LIN {X 0,Y 320.102,Z 625.92,A -85,B 0,C 180,E1 2193.671,E2 2193.671} C_VEL
LIN {X 0,Y 317.839,Z 623.977,A -85,B 0,C 180,E1 2191.692,E2 2191.692} C_VEL
LIN {X 0,Y 312.964,Z 620.611,A -85,B 0,C 180,E1 2187.803,E2 2187.803} C_VEL
LIN {X 0,Y 308.078,Z 616.466,A -85,B 0,C 180,E1 2184.137,E2 2184.137} C_VEL
LIN {X 0,Y 302.744,Z 613.332,A -85,B 0,C 180,E1 2180.694,E2 2180.694} C_VEL
LIN {X 0,Y 290.783,Z 600.623,A -85,B 0,C 180,E1 2170,E2 2170} C_VEL
LIN {X 0,Y 289.922,Z 598.567,A -85,B 0,C 180,E1 2168.424,E2 2168.424} C_VEL
LIN {X 0,Y 284.718,Z 621.095,A -85,B 0,C 180,E1 2168.26,E2 2168.26} C_VEL
LIN {X 0,Y 277.743,Z 643.252,A -85,B 0,C 180,E1 2168.127,E2 2168.127} C_VEL
LIN {X 0,Y 269.048,Z 664.747,A -85,B 0,C 180,E1 2167.961,E2 2167.961} C_VEL
LIN {X 0,Y 258.806,Z 685.28,A -85,B 0,C 180,E1 2167.727,E2 2167.727} C_VEL
LIN {X 0,Y 246.51,Z 705.546,A -85,B 0,C 180,E1 2167.398,E2 2167.398} C_VEL
LIN {X 0,Y 233.192,Z 724.08,A -85,B 0,C 180,E1 2166.987,E2 2166.987} C_VEL
LIN {X 0,Y 217.831,Z 742.232,A -85,B 0,C 180,E1 2166.425,E2 2166.425} C_VEL
LIN {X 0,Y 201.977,Z 758.277,A -85,B 0,C 180,E1 2165.734,E2 2165.734} C_VEL
LIN {X 0,Y 183.6,Z 774.186,A -85,B 0,C 180,E1 2164.75,E2 2164.75} C_VEL
LIN {X 0,Y 165.285,Z 787.803,A -85,B 0,C 180,E1 2163.525,E2 2163.525} C_VEL
LIN {X 0,Y 145.045,Z 800.516,A -85,B 0,C 180,E1 2161.78,E2 2161.78} C_VEL
LIN {X 0,Y 125.982,Z 810.635,A -85,B 0,C 180,E1 2159.595,E2 2159.595} C_VEL
LIN {X 0,Y 104.228,Z 820.309,A -85,B 0,C 180,E1 2156.063,E2 2156.063} C_VEL
LIN {X 0,Y 84.008,Z 827.603,A -85,B 0,C 180,E1 2151.055,E2 2151.055} C_VEL
LIN {X 0,Y 63.033,Z 833.661,A -85,B 0,C 180,E1 2142.124,E2 2142.124} C_VEL
LIN {X 0,Y 45.429,Z 837.544,A -85,B 0,C 180,E1 2126.617,E2 2126.617} C_VEL
LIN {X 0,Y 34.523,Z 839.63,A -85,B 0,C 180,E1 2101.419,E2 2101.419} C_VEL
LIN {X 0,Y 32.041,Z 840.272,A -85,B 0,C 180,E1 2073.061,E2 2073.061} C_VEL
LIN {X 0,Y 32.169,Z 840.12,A -85,B 0,C 180,E1 2057.434,E2 2057.434} C_VEL
LIN {X 0,Y 37.039,Z 839.124,A -85,B 0,C 180,E1 2029.62,E2 2029.62} C_VEL
LIN {X 0,Y 51.419,Z 836.361,A -85,B 0,C 180,E1 2006.561,E2 2006.561} C_VEL
LIN {X 0,Y 70.128,Z 831.753,A -85,B 0,C 180,E1 1994.188,E2 1994.188} C_VEL
LIN {X 0,Y 89.711,Z 825.717,A -85,B 0,C 180,E1 1987.293,E2 1987.293} C_VEL
LIN {X 0,Y 111.668,Z 817.214,A -85,B 0,C 180,E1 1982.566,E2 1982.566} C_VEL
LIN {X 0,Y 129.978,Z 808.641,A -85,B 0,C 180,E1 1979.893,E2 1979.893} C_VEL
LIN {X 0,Y 150.342,Z 797.394,A -85,B 0,C 180,E1 1977.713,E2 1977.713} C_VEL
LIN {X 0,Y 169.348,Z 784.933,A -85,B 0,C 180,E1 1976.176,E2 1976.176} C_VEL
LIN {X 0,Y 187.678,Z 770.939,A -85,B 0,C 180,E1 1975.014,E2 1975.014} C_VEL
LIN {X 0,Y 205.046,Z 755.352,A -85,B 0,C 180,E1 1974.123,E2 1974.123} C_VEL
LIN {X 0,Y 220.902,Z 738.824,A -85,B 0,C 180,E1 1973.455,E2 1973.455} C_VEL
LIN {X 0,Y 235.753,Z 720.694,A -85,B 0,C 180,E1 1972.929,E2 1972.929} C_VEL
LIN {X 0,Y 249.072,Z 701.604,A -85,B 0,C 180,E1 1972.53,E2 1972.53} C_VEL
LIN {X 0,Y 251.814,Z 697.259,A -85,B 0,C 180,E1 1972.457,E2 1972.457} C_VEL
LIN {X 0,Y 255.871,Z 690.789,A -85,B 0,C 180,E1 1972.136,E2 1972.136} C_VEL
LIN {X 0,Y 265.428,Z 674.452,A -85,B 0,C 180,E1 1970.638,E2 1970.638} C_VEL
LIN {X 0,Y 268.838,Z 667.606,A -85,B 0,C 180,E1 1970.369,E2 1970.369} C_VEL
LIN {X 0,Y 277.455,Z 647.28,A -85,B 0,C 180,E1 1970.258,E2 1970.258} C_VEL
LIN {X 0,Y 285.113,Z 624.081,A -85,B 0,C 180,E1 1970.163,E2 1970.163} C_VEL
LIN {X 0,Y 289.087,Z 608.609,A -85,B 0,C 180,E1 1970.042,E2 1970.042} C_VEL
LIN {X 0,Y 301.141,Z 621.43,A -85,B 0,C 180,E1 1958.987,E2 1958.987} C_VEL
LIN {X 0,Y 306.567,Z 624.761,A -85,B 0,C 180,E1 1955.428,E2 1955.428} C_VEL
LIN {X 0,Y 311.119,Z 628.561,A -85,B 0,C 180,E1 1952.017,E2 1952.017} C_VEL
LIN {X 0,Y 315.891,Z 631.757,A -85,B 0,C 180,E1 1948.303,E2 1948.303} C_VEL
LIN {X 0,Y 318.81,Z 634.401,A -85,B 0,C 180,E1 1945.74,E2 1945.74} C_VEL
LIN {X 0,Y 322.94,Z 637.822,A -85,B 0,C 180,E1 1941.966,E2 1941.966} C_VEL
LIN {X 0,Y 327.018,Z 640.577,A -85,B 0,C 180,E1 1938.082,E2 1938.082} C_VEL
LIN {X 0,Y 330.44,Z 644.079,A -85,B 0,C 180,E1 1934.343,E2 1934.343} C_VEL
LIN {X 0,Y 333.893,Z 646.67,A -85,B 0,C 180,E1 1930.482,E2 1930.482} C_VEL
LIN {X 0,Y 336.83,Z 648.45,A -85,B 0,C 180,E1 1927.012,E2 1927.012} C_VEL
LIN {X 0,Y 339.519,Z 651.579,A -85,B 0,C 180,E1 1923.212,E2 1923.212} C_VEL
LIN {X 0,Y 342.103,Z 653.743,A -85,B 0,C 180,E1 1919.406,E2 1919.406} C_VEL
LIN {X 0,Y 344.514,Z 655.168,A -85,B 0,C 180,E1 1915.499,E2 1915.499} C_VEL
LIN {X 0,Y 346.58,Z 656.053,A -85,B 0,C 180,E1 1911.729,E2 1911.729} C_VEL
LIN {X 0,Y 348.102,Z 658.201,A -85,B 0,C 180,E1 1907.898,E2 1907.898} C_VEL
LIN {X 0,Y 349.354,Z 659.732,A -85,B 0,C 180,E1 1904.248,E2 1904.248} C_VEL
LIN {X 0,Y 350.337,Z 660.737,A -85,B 0,C 180,E1 1900.524,E2 1900.524} C_VEL
LIN {X 0,Y 351.081,Z 661.354,A -85,B 0,C 180,E1 1896.705,E2 1896.705} C_VEL
LIN {X 0,Y 351.475,Z 661.618,A -85,B 0,C 180,E1 1893.135,E2 1893.135} C_VEL
LIN {X 0,Y 351.583,Z 661.704,A -85,B 0,C 180,E1 1889.348,E2 1889.348} C_VEL
LIN {X 0,Y 351.381,Z 661.597,A -85,B 0,C 180,E1 1885.921,E2 1885.921} C_VEL
LIN {X 0,Y 350.894,Z 661.181,A -85,B 0,C 180,E1 1882.139,E2 1882.139} C_VEL
LIN {X 0,Y 350.09,Z 660.488,A -85,B 0,C 180,E1 1878.409,E2 1878.409} C_VEL
LIN {X 0,Y 349.022,Z 659.363,A -85,B 0,C 180,E1 1874.719,E2 1874.719} C_VEL
LIN {X 0,Y 347.649,Z 657.577,A -85,B 0,C 180,E1 1870.861,E2 1870.861} C_VEL
LIN {X 0,Y 346.392,Z 655.984,A -85,B 0,C 180,E1 1867.905,E2 1867.905} C_VEL
LIN {X 0,Y 344.411,Z 655.129,A -85,B 0,C 180,E1 1864.371,E2 1864.371} C_VEL
LIN {X 0,Y 341.976,Z 653.652,A -85,B 0,C 180,E1 1860.389,E2 1860.389} C_VEL
LIN {X 0,Y 339.315,Z 651.382,A -85,B 0,C 180,E1 1856.503,E2 1856.503} C_VEL
LIN {X 0,Y 336.812,Z 648.412,A -85,B 0,C 180,E1 1852.943,E2 1852.943} C_VEL
LIN {X 0,Y 333.403,Z 646.352,A -85,B 0,C 180,E1 1848.947,E2 1848.947} C_VEL
LIN {X 0,Y 330.101,Z 643.814,A -85,B 0,C 180,E1 1845.356,E2 1845.356} C_VEL
LIN {X 0,Y 327.244,Z 640.903,A -85,B 0,C 180,E1 1842.236,E2 1842.236} C_VEL
LIN {X 0,Y 325.416,Z 639.465,A -85,B 0,C 180,E1 1840.362,E2 1840.362} C_VEL
LIN {X 0,Y 321.239,Z 636.539,A -85,B 0,C 180,E1 1836.476,E2 1836.476} C_VEL
LIN {X 0,Y 317.034,Z 632.556,A -85,B 0,C 180,E1 1832.636,E2 1832.636} C_VEL
LIN {X 0,Y 312.081,Z 629.265,A -85,B 0,C 180,E1 1828.723,E2 1828.723} C_VEL
LIN {X 0,Y 307.338,Z 625.454,A -85,B 0,C 180,E1 1825.122,E2 1825.122} C_VEL
LIN {X 0,Y 304.559,Z 623.461,A -85,B 0,C 180,E1 1823.201,E2 1823.201} C_VEL
LIN {X 0,Y 298.441,Z 619.537,A -85,B 0,C 180,E1 1819.269,E2 1819.269} C_VEL
LIN {X 0,Y 291.516,Z 612.567,A -85,B 0,C 180,E1 1813.285,E2 1813.285} C_VEL
LIN {X 0,Y 289.022,Z 608.749,A -85,B 0,C 180,E1 1809.919,E2 1809.919} C_VEL
LIN {X 0,Y 282.774,Z 631.763,A -85,B 0,C 180,E1 1809.809,E2 1809.809} C_VEL
LIN {X 0,Y 274.898,Z 653.734,A -85,B 0,C 180,E1 1809.717,E2 1809.717} C_VEL
LIN {X 0,Y 265.662,Z 674.23,A -85,B 0,C 180,E1 1809.583,E2 1809.583} C_VEL
LIN {X 0,Y 255.391,Z 693.035,A -85,B 0,C 180,E1 1809.406,E2 1809.406} C_VEL
LIN {X 0,Y 242.675,Z 712.598,A -85,B 0,C 180,E1 1809.148,E2 1809.148} C_VEL
LIN {X 0,Y 228.664,Z 730.782,A -85,B 0,C 180,E1 1808.817,E2 1808.817} C_VEL
LIN {X 0,Y 213.039,Z 748.159,A -85,B 0,C 180,E1 1808.366,E2 1808.366} C_VEL
LIN {X 0,Y 196.79,Z 763.614,A -85,B 0,C 180,E1 1807.806,E2 1807.806} C_VEL
LIN {X 0,Y 180.354,Z 777.15,A -85,B 0,C 180,E1 1807.104,E2 1807.104} C_VEL
LIN {X 0,Y 160.873,Z 790.935,A -85,B 0,C 180,E1 1806.065,E2 1806.065} C_VEL
LIN {X 0,Y 140.436,Z 803.092,A -85,B 0,C 180,E1 1804.64,E2 1804.64} C_VEL
LIN {X 0,Y 119.102,Z 813.711,A -85,B 0,C 180,E1 1802.598,E2 1802.598} C_VEL
LIN {X 0,Y 98.984,Z 821.939,A -85,B 0,C 180,E1 1799.842,E2 1799.842} C_VEL
LIN {X 0,Y 77.255,Z 829.128,A -85,B 0,C 180,E1 1795.222,E2 1795.222} C_VEL
LIN {X 0,Y 56.371,Z 834.404,A -85,B 0,C 180,E1 1787.294,E2 1787.294} C_VEL
LIN {X 0,Y 38.335,Z 837.829,A -85,B 0,C 180,E1 1772.469,E2 1772.469} C_VEL
LIN {X 0,Y 25.468,Z 839.709,A -85,B 0,C 180,E1 1738.106,E2 1738.106} C_VEL
LIN {X 0,Y 24.077,Z 840.061,A -85,B 0,C 180,E1 1710,E2 1710} C_VEL
LIN {X 0,Y 26.34,Z 839.628,A -85,B 0,C 180,E1 1676.629,E2 1676.629} C_VEL
LIN {X 0,Y 39.907,Z 837.567,A -85,B 0,C 180,E1 1645.587,E2 1645.587} C_VEL
LIN {X 0,Y 58.213,Z 834.008,A -85,B 0,C 180,E1 1631.765,E2 1631.765} C_VEL
LIN {X 0,Y 80.183,Z 828.281,A -85,B 0,C 180,E1 1624.009,E2 1624.009} C_VEL
LIN {X 0,Y 101.984,Z 820.822,A -85,B 0,C 180,E1 1619.678,E2 1619.678} C_VEL
LIN {X 0,Y 124.166,Z 811.372,A -85,B 0,C 180,E1 1616.851,E2 1616.851} C_VEL
LIN {X 0,Y 143.496,Z 801.397,A -85,B 0,C 180,E1 1615.12,E2 1615.12} C_VEL
LIN {X 0,Y 162.922,Z 789.581,A -85,B 0,C 180,E1 1613.812,E2 1613.812} C_VEL
LIN {X 0,Y 182.408,Z 775.547,A -85,B 0,C 180,E1 1612.799,E2 1612.799} C_VEL
LIN {X 0,Y 200.186,Z 760.621,A -85,B 0,C 180,E1 1612.067,E2 1612.067} C_VEL
LIN {X 0,Y 217.352,Z 743.64,A -85,B 0,C 180,E1 1611.498,E2 1611.498} C_VEL
LIN {X 0,Y 232.362,Z 726.314,A -85,B 0,C 180,E1 1611.089,E2 1611.089} C_VEL
LIN {X 0,Y 246.142,Z 707.607,A -85,B 0,C 180,E1 1610.776,E2 1610.776} C_VEL
LIN {X 0,Y 257.962,Z 688.601,A -85,B 0,C 180,E1 1610.544,E2 1610.544} C_VEL
LIN {X 0,Y 268.838,Z 667.606,A -85,B 0,C 180,E1 1610.369,E2 1610.369} C_VEL
LIN {X 0,Y 272.169,Z 660.669,A -85,B 0,C 180,E1 1610.127,E2 1610.127} C_VEL
LIN {X 0,Y 280.144,Z 643.301,A -85,B 0,C 180,E1 1608.817,E2 1608.817} C_VEL
LIN {X 0,Y 282.804,Z 636.101,A -85,B 0,C 180,E1 1608.603,E2 1608.603} C_VEL
LIN {X 0,Y 288.084,Z 618.389,A -85,B 0,C 180,E1 1608.544,E2 1608.544} C_VEL
LIN {X 0,Y 292.739,Z 624.151,A -85,B 0,C 180,E1 1603.429,E2 1603.429} C_VEL
LIN {X 0,Y 301.039,Z 630.48,A -85,B 0,C 180,E1 1597.545,E2 1597.545} C_VEL
LIN {X 0,Y 304.376,Z 632.619,A -85,B 0,C 180,E1 1595.343,E2 1595.343} C_VEL
LIN {X 0,Y 309.353,Z 636.641,A -85,B 0,C 180,E1 1591.633,E2 1591.633} C_VEL
LIN {X 0,Y 314.36,Z 639.845,A -85,B 0,C 180,E1 1587.781,E2 1587.781} C_VEL
LIN {X 0,Y 318.543,Z 643.821,A -85,B 0,C 180,E1 1584.058,E2 1584.058} C_VEL
LIN {X 0,Y 322.898,Z 646.911,A -85,B 0,C 180,E1 1580.135,E2 1580.135} C_VEL
LIN {X 0,Y 325.225,Z 648.595,A -85,B 0,C 180,E1 1577.917,E2 1577.917} C_VEL
LIN {X 0,Y 328.789,Z 652.073,A -85,B 0,C 180,E1 1574.137,E2 1574.137} C_VEL
LIN {X 0,Y 332.304,Z 654.586,A -85,B 0,C 180,E1 1570.307,E2 1570.307} C_VEL
LIN {X 0,Y 335.15,Z 656.305,A -85,B 0,C 180,E1 1567.057,E2 1567.057} C_VEL
LIN {X 0,Y 337.799,Z 659.322,A -85,B 0,C 180,E1 1563.403,E2 1563.403} C_VEL
LIN {X 0,Y 340.461,Z 661.535,A -85,B 0,C 180,E1 1559.562,E2 1559.562} C_VEL
LIN {X 0,Y 342.896,Z 662.969,A -85,B 0,C 180,E1 1555.751,E2 1555.751} C_VEL
LIN {X 0,Y 345.097,Z 663.894,A -85,B 0,C 180,E1 1551.947,E2 1551.947} C_VEL
LIN {X 0,Y 346.625,Z 665.9,A -85,B 0,C 180,E1 1548.325,E2 1548.325} C_VEL
LIN {X 0,Y 347.922,Z 667.484,A -85,B 0,C 180,E1 1544.648,E2 1544.648} C_VEL
LIN {X 0,Y 348.994,Z 668.566,A -85,B 0,C 180,E1 1540.899,E2 1540.899} C_VEL
LIN {X 0,Y 349.798,Z 669.201,A -85,B 0,C 180,E1 1537.06,E2 1537.06} C_VEL
LIN {X 0,Y 350.268,Z 669.523,A -85,B 0,C 180,E1 1533.273,E2 1533.273} C_VEL
LIN {X 0,Y 350.374,Z 669.619,A -85,B 0,C 180,E1 1529.509,E2 1529.509} C_VEL
LIN {X 0,Y 350.147,Z 669.5,A -85,B 0,C 180,E1 1525.906,E2 1525.906} C_VEL
LIN {X 0,Y 349.635,Z 669.089,A -85,B 0,C 180,E1 1522.276,E2 1522.276} C_VEL
LIN {X 0,Y 348.813,Z 668.434,A -85,B 0,C 180,E1 1518.593,E2 1518.593} C_VEL
LIN {X 0,Y 347.755,Z 667.302,A -85,B 0,C 180,E1 1514.833,E2 1514.833} C_VEL
LIN {X 0,Y 346.421,Z 665.635,A -85,B 0,C 180,E1 1511.14,E2 1511.14} C_VEL
LIN {X 0,Y 345.072,Z 663.886,A -85,B 0,C 180,E1 1508.004,E2 1508.004} C_VEL
LIN {X 0,Y 342.801,Z 662.921,A -85,B 0,C 180,E1 1504.056,E2 1504.056} C_VEL
LIN {X 0,Y 340.303,Z 661.435,A -85,B 0,C 180,E1 1500.229,E2 1500.229} C_VEL
LIN {X 0,Y 337.633,Z 659.166,A -85,B 0,C 180,E1 1496.375,E2 1496.375} C_VEL
LIN {X 0,Y 334.789,Z 655.876,A -85,B 0,C 180,E1 1492.466,E2 1492.466} C_VEL
LIN {X 0,Y 331.341,Z 653.985,A -85,B 0,C 180,E1 1488.636,E2 1488.636} C_VEL
LIN {X 0,Y 327.939,Z 651.333,A -85,B 0,C 180,E1 1484.982,E2 1484.982} C_VEL
LIN {X 0,Y 324.58,Z 647.915,A -85,B 0,C 180,E1 1481.475,E2 1481.475} C_VEL
LIN {X 0,Y 320.732,Z 645.471,A -85,B 0,C 180,E1 1477.889,E2 1477.889} C_VEL
LIN {X 0,Y 316.383,Z 641.914,A -85,B 0,C 180,E1 1474.012,E2 1474.012} C_VEL
LIN {X 0,Y 313.673,Z 639.451,A -85,B 0,C 180,E1 1471.673,E2 1471.673} C_VEL
LIN {X 0,Y 308.376,Z 635.921,A -85,B 0,C 180,E1 1467.623,E2 1467.623} C_VEL
LIN {X 0,Y 303.057,Z 631.562,A -85,B 0,C 180,E1 1463.735,E2 1463.735} C_VEL
LIN {X 0,Y 297.543,Z 628.3,A -85,B 0,C 180,E1 1460.25,E2 1460.25} C_VEL
LIN {X 0,Y 288.077,Z 618.375,A -85,B 0,C 180,E1 1451.445,E2 1451.445} C_VEL
LIN {X 0,Y 280.983,Z 641.308,A -85,B 0,C 180,E1 1451.386,E2 1451.386} C_VEL
LIN {X 0,Y 272.778,Z 662,A -85,B 0,C 180,E1 1451.338,E2 1451.338} C_VEL
LIN {X 0,Y 263.015,Z 681.892,A -85,B 0,C 180,E1 1451.255,E2 1451.255} C_VEL
LIN {X 0,Y 250.661,Z 702.717,A -85,B 0,C 180,E1 1451.116,E2 1451.116} C_VEL
LIN {X 0,Y 237.784,Z 720.866,A -85,B 0,C 180,E1 1450.943,E2 1450.943} C_VEL
LIN {X 0,Y 222.317,Z 739.456,A -85,B 0,C 180,E1 1450.684,E2 1450.684} C_VEL
LIN {X 0,Y 205.993,Z 756.147,A -85,B 0,C 180,E1 1450.346,E2 1450.346} C_VEL
LIN {X 0,Y 187.747,Z 772.052,A -85,B 0,C 180,E1 1449.87,E2 1449.87} C_VEL
LIN {X 0,Y 169.173,Z 785.863,A -85,B 0,C 180,E1 1449.253,E2 1449.253} C_VEL
LIN {X 0,Y 148.553,Z 798.868,A -85,B 0,C 180,E1 1448.36,E2 1448.36} C_VEL
LIN {X 0,Y 128.146,Z 809.543,A -85,B 0,C 180,E1 1447.171,E2 1447.171} C_VEL
LIN {X 0,Y 106.436,Z 819.024,A -85,B 0,C 180,E1 1445.39,E2 1445.39} C_VEL
LIN {X 0,Y 84.774,Z 826.564,A -85,B 0,C 180,E1 1442.704,E2 1442.704} C_VEL
LIN {X 0,Y 62.937,Z 832.47,A -85,B 0,C 180,E1 1438.179,E2 1438.179} C_VEL
LIN {X 0,Y 40.786,Z 836.743,A -85,B 0,C 180,E1 1428.682,E2 1428.682} C_VEL
LIN {X 0,Y 23.694,Z 838.961,A -85,B 0,C 180,E1 1407.559,E2 1407.559} C_VEL
LIN {X 0,Y 16.042,Z 839.766,A -85,B 0,C 180,E1 1357.161,E2 1357.161} C_VEL
LIN {X 0,Y 16.174,Z 839.709,A -85,B 0,C 180,E1 1335.684,E2 1335.684} C_VEL
LIN {X 0,Y 25.189,Z 838.794,A -85,B 0,C 180,E1 1289.163,E2 1289.163} C_VEL
LIN {X 0,Y 43.599,Z 836.315,A -85,B 0,C 180,E1 1269.568,E2 1269.568} C_VEL
LIN {X 0,Y 66.589,Z 831.602,A -85,B 0,C 180,E1 1260.86,E2 1260.86} C_VEL
LIN {X 0,Y 89.137,Z 825.198,A -85,B 0,C 180,E1 1256.651,E2 1256.651} C_VEL
LIN {X 0,Y 111.567,Z 816.952,A -85,B 0,C 180,E1 1254.127,E2 1254.127} C_VEL
LIN {X 0,Y 131.059,Z 808.13,A -85,B 0,C 180,E1 1252.634,E2 1252.634} C_VEL
LIN {X 0,Y 151.645,Z 797.029,A -85,B 0,C 180,E1 1251.487,E2 1251.487} C_VEL
LIN {X 0,Y 171.236,Z 784.428,A -85,B 0,C 180,E1 1250.671,E2 1250.671} C_VEL
LIN {X 0,Y 189.81,Z 770.429,A -85,B 0,C 180,E1 1250.072,E2 1250.072} C_VEL
LIN {X 0,Y 207.356,Z 754.855,A -85,B 0,C 180,E1 1249.625,E2 1249.625} C_VEL
LIN {X 0,Y 223.348,Z 738.314,A -85,B 0,C 180,E1 1249.297,E2 1249.297} C_VEL
LIN {X 0,Y 238.299,Z 720.189,A -85,B 0,C 180,E1 1249.05,E2 1249.05} C_VEL
LIN {X 0,Y 251.691,Z 701.094,A -85,B 0,C 180,E1 1248.871,E2 1248.871} C_VEL
LIN {X 0,Y 263.528,Z 680.907,A -85,B 0,C 180,E1 1248.74,E2 1248.74} C_VEL
LIN {X 0,Y 273.29,Z 660.869,A -85,B 0,C 180,E1 1248.659,E2 1248.659} C_VEL
LIN {X 0,Y 282.009,Z 638.446,A -85,B 0,C 180,E1 1248.608,E2 1248.608} C_VEL
LIN {X 0,Y 282.804,Z 636.101,A -85,B 0,C 180,E1 1248.603,E2 1248.603} C_VEL
LIN {X 0,Y 283.769,Z 633.683,A -85,B 0,C 180,E1 1248.417,E2 1248.417} C_VEL
LIN {X 0,Y 285.071,Z 631.417,A -85,B 0,C 180,E1 1247.845,E2 1247.845} C_VEL
LIN {X 0,Y 286.72,Z 629.9,A -85,B 0,C 180,E1 1246.763,E2 1246.763} C_VEL
LIN {X 0,Y 288.308,Z 630.127,A -85,B 0,C 180,E1 1245.362,E2 1245.362} C_VEL
LIN {X 0,Y 292.182,Z 633.688,A -85,B 0,C 180,E1 1241.856,E2 1241.856} C_VEL
LIN {X 0,Y 299.648,Z 638.71,A -85,B 0,C 180,E1 1236.813,E2 1236.813} C_VEL
LIN {X 0,Y 303.358,Z 641.604,A -85,B 0,C 180,E1 1234.211,E2 1234.211} C_VEL
LIN {X 0,Y 308.38,Z 645.33,A -85,B 0,C 180,E1 1230.473,E2 1230.473} C_VEL
LIN {X 0,Y 312.275,Z 647.928,A -85,B 0,C 180,E1 1227.459,E2 1227.459} C_VEL
LIN {X 0,Y 316.501,Z 651.746,A -85,B 0,C 180,E1 1223.79,E2 1223.79} C_VEL
LIN {X 0,Y 320.979,Z 654.789,A -85,B 0,C 180,E1 1219.849,E2 1219.849} C_VEL
LIN {X 0,Y 322.945,Z 656.276,A -85,B 0,C 180,E1 1217.991,E2 1217.991} C_VEL
LIN {X 0,Y 326.545,Z 659.732,A -85,B 0,C 180,E1 1214.235,E2 1214.235} C_VEL
LIN {X 0,Y 330.211,Z 662.294,A -85,B 0,C 180,E1 1210.388,E2 1210.388} C_VEL
LIN {X 0,Y 333.151,Z 664.081,A -85,B 0,C 180,E1 1207.101,E2 1207.101} C_VEL
LIN {X 0,Y 336.035,Z 667.258,A -85,B 0,C 180,E1 1203.194,E2 1203.194} C_VEL
LIN {X 0,Y 338.775,Z 669.429,A -85,B 0,C 180,E1 1199.335,E2 1199.335} C_VEL
LIN {X 0,Y 341.183,Z 670.791,A -85,B 0,C 180,E1 1195.703,E2 1195.703} C_VEL
LIN {X 0,Y 343.504,Z 671.748,A -85,B 0,C 180,E1 1191.793,E2 1191.793} C_VEL
LIN {X 0,Y 345.075,Z 673.879,A -85,B 0,C 180,E1 1188.061,E2 1188.061} C_VEL
LIN {X 0,Y 346.366,Z 675.429,A -85,B 0,C 180,E1 1184.374,E2 1184.374} C_VEL
LIN {X 0,Y 347.439,Z 676.46,A -85,B 0,C 180,E1 1180.613,E2 1180.613} C_VEL
LIN {X 0,Y 348.22,Z 677.066,A -85,B 0,C 180,E1 1176.926,E2 1176.926} C_VEL
LIN {X 0,Y 348.709,Z 677.369,A -85,B 0,C 180,E1 1173.287,E2 1173.287} C_VEL
LIN {X 0,Y 348.818,Z 677.467,A -85,B 0,C 180,E1 1169.507,E2 1169.507} C_VEL
LIN {X 0,Y 348.578,Z 677.344,A -85,B 0,C 180,E1 1165.888,E2 1165.888} C_VEL
LIN {X 0,Y 348.047,Z 676.928,A -85,B 0,C 180,E1 1162.24,E2 1162.24} C_VEL
LIN {X 0,Y 347.207,Z 676.265,A -85,B 0,C 180,E1 1158.539,E2 1158.539} C_VEL
LIN {X 0,Y 346.104,Z 675.121,A -85,B 0,C 180,E1 1154.772,E2 1154.772} C_VEL
LIN {X 0,Y 344.762,Z 673.44,A -85,B 0,C 180,E1 1151.046,E2 1151.046} C_VEL
LIN {X 0,Y 343.315,Z 671.678,A -85,B 0,C 180,E1 1147.839,E2 1147.839} C_VEL
LIN {X 0,Y 340.832,Z 670.628,A -85,B 0,C 180,E1 1143.707,E2 1143.707} C_VEL
LIN {X 0,Y 338.304,Z 669.12,A -85,B 0,C 180,E1 1139.992,E2 1139.992} C_VEL
LIN {X 0,Y 335.565,Z 666.801,A -85,B 0,C 180,E1 1136.139,E2 1136.139} C_VEL
LIN {X 0,Y 332.576,Z 663.521,A -85,B 0,C 180,E1 1132.172,E2 1132.172} C_VEL
LIN {X 0,Y 329.045,Z 661.572,A -85,B 0,C 180,E1 1128.375,E2 1128.375} C_VEL
LIN {X 0,Y 325.334,Z 658.656,A -85,B 0,C 180,E1 1124.484,E2 1124.484} C_VEL
LIN {X 0,Y 321.642,Z 655.159,A -85,B 0,C 180,E1 1120.753,E2 1120.753} C_VEL
LIN {X 0,Y 317.407,Z 652.426,A -85,B 0,C 180,E1 1116.989,E2 1116.989} C_VEL
LIN {X 0,Y 312.962,Z 648.617,A -85,B 0,C 180,E1 1113.114,E2 1113.114} C_VEL
LIN {X 0,Y 310.633,Z 646.739,A -85,B 0,C 180,E1 1111.213,E2 1111.213} C_VEL
LIN {X 0,Y 305.618,Z 643.387,A -85,B 0,C 180,E1 1107.471,E2 1107.471} C_VEL
LIN {X 0,Y 300.715,Z 639.279,A -85,B 0,C 180,E1 1103.889,E2 1103.889} C_VEL
LIN {X 0,Y 294.474,Z 635.528,A -85,B 0,C 180,E1 1099.849,E2 1099.849} C_VEL
LIN {X 0,Y 286.992,Z 627.863,A -85,B 0,C 180,E1 1092.986,E2 1092.986} C_VEL
LIN {X 0,Y 279.601,Z 649.44,A -85,B 0,C 180,E1 1092.983,E2 1092.983} C_VEL
LIN {X 0,Y 270.875,Z 669.52,A -85,B 0,C 180,E1 1092.979,E2 1092.979} C_VEL
LIN {X 0,Y 260.076,Z 689.881,A -85,B 0,C 180,E1 1092.954,E2 1092.954} C_VEL
LIN {X 0,Y 247.709,Z 709.32,A -85,B 0,C 180,E1 1092.898,E2 1092.898} C_VEL
LIN {X 0,Y 233.268,Z 728.413,A -85,B 0,C 180,E1 1092.811,E2 1092.811} C_VEL
LIN {X 0,Y 218.288,Z 745.346,A -85,B 0,C 180,E1 1092.68,E2 1092.68} C_VEL
LIN {X 0,Y 200.711,Z 762.216,A -85,B 0,C 180,E1 1092.483,E2 1092.483} C_VEL
LIN {X 0,Y 184.052,Z 775.92,A -85,B 0,C 180,E1 1092.232,E2 1092.232} C_VEL
LIN {X 0,Y 164.477,Z 789.741,A -85,B 0,C 180,E1 1091.848,E2 1091.848} C_VEL
LIN {X 0,Y 143.763,Z 802.022,A -85,B 0,C 180,E1 1091.301,E2 1091.301} C_VEL
LIN {X 0,Y 122.026,Z 812.755,A -85,B 0,C 180,E1 1090.508,E2 1090.508} C_VEL
LIN {X 0,Y 101.352,Z 821.056,A -85,B 0,C 180,E1 1089.427,E2 1089.427} C_VEL
LIN {X 0,Y 78.681,Z 828.326,A -85,B 0,C 180,E1 1087.619,E2 1087.619} C_VEL
LIN {X 0,Y 56.165,Z 833.697,A -85,B 0,C 180,E1 1084.514,E2 1084.514} C_VEL
LIN {X 0,Y 35.009,Z 837.185,A -85,B 0,C 180,E1 1078.35,E2 1078.35} C_VEL
LIN {X 0,Y 14.274,Z 839.174,A -85,B 0,C 180,E1 1055.148,E2 1055.148} C_VEL
LIN {X 0,Y 8.059,Z 839.563,A -85,B 0,C 180,E1 990,E2 990} C_VEL
LIN {X 0,Y 17.766,Z 838.947,A -85,B 0,C 180,E1 916.919,E2 916.919} C_VEL
LIN {X 0,Y 37.994,Z 836.774,A -85,B 0,C 180,E1 900.39,E2 900.39} C_VEL
LIN {X 0,Y 61.262,Z 832.653,A -85,B 0,C 180,E1 894.597,E2 894.597} C_VEL
LIN {X 0,Y 84.469,Z 826.642,A -85,B 0,C 180,E1 891.834,E2 891.834} C_VEL
LIN {X 0,Y 105.483,Z 819.532,A -85,B 0,C 180,E1 890.322,E2 890.322} C_VEL
LIN {X 0,Y 128.415,Z 809.778,A -85,B 0,C 180,E1 889.23,E2 889.23} C_VEL
LIN {X 0,Y 147.906,Z 799.753,A -85,B 0,C 180,E1 888.575,E2 888.575} C_VEL
LIN {X 0,Y 169.052,Z 786.745,A -85,B 0,C 180,E1 888.053,E2 888.053} C_VEL
LIN {X 0,Y 187.822,Z 772.978,A -85,B 0,C 180,E1 887.705,E2 887.705} C_VEL
LIN {X 0,Y 205.883,Z 757.51,A -85,B 0,C 180,E1 887.453,E2 887.453} C_VEL
LIN {X 0,Y 222.502,Z 740.823,A -85,B 0,C 180,E1 887.28,E2 887.28} C_VEL
LIN {X 0,Y 237.91,Z 722.645,A -85,B 0,C 180,E1 887.159,E2 887.159} C_VEL
LIN {X 0,Y 251.317,Z 704.037,A -85,B 0,C 180,E1 887.084,E2 887.084} C_VEL
LIN {X 0,Y 263.678,Z 683.61,A -85,B 0,C 180,E1 887.035,E2 887.035} C_VEL
LIN {X 0,Y 273.961,Z 662.886,A -85,B 0,C 180,E1 887.014,E2 887.014} C_VEL
LIN {X 0,Y 282.424,Z 641.766,A -85,B 0,C 180,E1 887.016,E2 887.016} C_VEL
LIN {X 0,Y 286.991,Z 627.863,A -85,B 0,C 180,E1 887.014,E2 887.014} C_VEL
LIN {X 0,Y 292.182,Z 633.688,A -85,B 0,C 180,E1 881.856,E2 881.856} C_VEL
LIN {X 0,Y 293.962,Z 636.519,A -85,B 0,C 180,E1 880.252,E2 880.252} C_VEL
LIN {X 0,Y 297.382,Z 645.819,A -85,B 0,C 180,E1 876.617,E2 876.617} C_VEL
LIN {X 0,Y 298.597,Z 647.472,A -85,B 0,C 180,E1 875.623,E2 875.623} C_VEL
LIN {X 0,Y 303.425,Z 651.344,A -85,B 0,C 180,E1 872.101,E2 872.101} C_VEL
LIN {X 0,Y 308.028,Z 654.336,A -85,B 0,C 180,E1 868.711,E2 868.711} C_VEL
LIN {X 0,Y 310.844,Z 656.749,A -85,B 0,C 180,E1 866.41,E2 866.41} C_VEL
LIN {X 0,Y 315.402,Z 660.432,A -85,B 0,C 180,E1 862.507,E2 862.507} C_VEL
LIN {X 0,Y 319.979,Z 663.395,A -85,B 0,C 180,E1 858.513,E2 858.513} C_VEL
LIN {X 0,Y 323.684,Z 666.992,A -85,B 0,C 180,E1 854.727,E2 854.727} C_VEL
LIN {X 0,Y 327.248,Z 669.574,A -85,B 0,C 180,E1 851.063,E2 851.063} C_VEL
LIN {X 0,Y 330.671,Z 671.513,A -85,B 0,C 180,E1 847.427,E2 847.427} C_VEL
LIN {X 0,Y 333.495,Z 674.645,A -85,B 0,C 180,E1 843.686,E2 843.686} C_VEL
LIN {X 0,Y 336.218,Z 676.862,A -85,B 0,C 180,E1 839.973,E2 839.973} C_VEL
LIN {X 0,Y 338.908,Z 678.425,A -85,B 0,C 180,E1 836.077,E2 836.077} C_VEL
LIN {X 0,Y 341.3,Z 679.414,A -85,B 0,C 180,E1 832.22,E2 832.22} C_VEL
LIN {X 0,Y 342.598,Z 680.961,A -85,B 0,C 180,E1 829.432,E2 829.432} C_VEL
LIN {X 0,Y 344.057,Z 682.748,A -85,B 0,C 180,E1 825.68,E2 825.68} C_VEL
LIN {X 0,Y 345.256,Z 683.951,A -85,B 0,C 180,E1 821.807,E2 821.807} C_VEL
LIN {X 0,Y 346.102,Z 684.675,A -85,B 0,C 180,E1 818.138,E2 818.138} C_VEL
LIN {X 0,Y 346.659,Z 685.093,A -85,B 0,C 180,E1 814.466,E2 814.466} C_VEL
LIN {X 0,Y 346.92,Z 685.227,A -85,B 0,C 180,E1 810.826,E2 810.826} C_VEL
LIN {X 0,Y 346.873,Z 685.183,A -85,B 0,C 180,E1 807.191,E2 807.191} C_VEL
LIN {X 0,Y 346.408,Z 684.909,A -85,B 0,C 180,E1 803.537,E2 803.537} C_VEL
LIN {X 0,Y 345.679,Z 684.324,A -85,B 0,C 180,E1 800.006,E2 800.006} C_VEL
LIN {X 0,Y 344.598,Z 683.362,A -85,B 0,C 180,E1 796.065,E2 796.065} C_VEL
LIN {X 0,Y 343.336,Z 681.89,A -85,B 0,C 180,E1 792.371,E2 792.371} C_VEL
LIN {X 0,Y 341.802,Z 679.787,A -85,B 0,C 180,E1 788.733,E2 788.733} C_VEL
LIN {X 0,Y 339.802,Z 678.831,A -85,B 0,C 180,E1 785.303,E2 785.303} C_VEL
LIN {X 0,Y 337.267,Z 677.507,A -85,B 0,C 180,E1 781.492,E2 781.492} C_VEL
LIN {X 0,Y 334.661,Z 675.64,A -85,B 0,C 180,E1 777.873,E2 777.873} C_VEL
LIN {X 0,Y 331.694,Z 672.728,A -85,B 0,C 180,E1 773.887,E2 773.887} C_VEL
LIN {X 0,Y 330.017,Z 671.061,A -85,B 0,C 180,E1 771.827,E2 771.827} C_VEL
LIN {X 0,Y 326.198,Z 668.899,A -85,B 0,C 180,E1 767.836,E2 767.836} C_VEL
LIN {X 0,Y 322.243,Z 665.699,A -85,B 0,C 180,E1 763.783,E2 763.783} C_VEL
LIN {X 0,Y 318.882,Z 662.615,A -85,B 0,C 180,E1 760.47,E2 760.47} C_VEL
LIN {X 0,Y 313.803,Z 659.262,A -85,B 0,C 180,E1 756.118,E2 756.118} C_VEL
LIN {X 0,Y 309.504,Z 655.424,A -85,B 0,C 180,E1 752.43,E2 752.43} C_VEL
LIN {X 0,Y 304.489,Z 652.077,A -85,B 0,C 180,E1 748.648,E2 748.648} C_VEL
LIN {X 0,Y 299.064,Z 647.879,A -85,B 0,C 180,E1 744.703,E2 744.703} C_VEL
LIN {X 0,Y 296.262,Z 645.902,A -85,B 0,C 180,E1 742.837,E2 742.837} C_VEL
LIN {X 0,Y 287.713,Z 639.519,A -85,B 0,C 180,E1 736.557,E2 736.557} C_VEL
LIN {X 0,Y 285.915,Z 637.121,A -85,B 0,C 180,E1 734.557,E2 734.557} C_VEL
LIN {X 0,Y 277.217,Z 659.694,A -85,B 0,C 180,E1 734.609,E2 734.609} C_VEL
LIN {X 0,Y 267.665,Z 679.421,A -85,B 0,C 180,E1 734.656,E2 734.656} C_VEL
LIN {X 0,Y 255.826,Z 699.772,A -85,B 0,C 180,E1 734.695,E2 734.695} C_VEL
LIN {X 0,Y 242.325,Z 719.137,A -85,B 0,C 180,E1 734.727,E2 734.727} C_VEL
LIN {X 0,Y 227.456,Z 737.233,A -85,B 0,C 180,E1 734.748,E2 734.748} C_VEL
LIN {X 0,Y 211.429,Z 753.858,A -85,B 0,C 180,E1 734.747,E2 734.747} C_VEL
LIN {X 0,Y 194.352,Z 769.064,A -85,B 0,C 180,E1 734.725,E2 734.725} C_VEL
LIN {X 0,Y 175.696,Z 783.206,A -85,B 0,C 180,E1 734.666,E2 734.666} C_VEL
LIN {X 0,Y 155.988,Z 795.899,A -85,B 0,C 180,E1 734.567,E2 734.567} C_VEL
LIN {X 0,Y 135.228,Z 807.119,A -85,B 0,C 180,E1 734.403,E2 734.403} C_VEL
LIN {X 0,Y 115.496,Z 816.007,A -85,B 0,C 180,E1 734.173,E2 734.173} C_VEL
LIN {X 0,Y 92.337,Z 824.447,A -85,B 0,C 180,E1 733.782,E2 733.782} C_VEL
LIN {X 0,Y 69.838,Z 830.734,A -85,B 0,C 180,E1 733.214,E2 733.214} C_VEL
LIN {X 0,Y 46.044,Z 835.507,A -85,B 0,C 180,E1 732.269,E2 732.269} C_VEL
LIN {X 0,Y 23.404,Z 838.2,A -85,B 0,C 180,E1 730.711,E2 730.711} C_VEL
LIN {X 0,Y 5.044,Z 839.177,A -85,B 0,C 180,E1 727.62,E2 727.62} C_VEL
LIN {X 0,Y 1.002,Z 839.294,A -85,B 0,C 180,E1 896.485,E2 896.485} C_VEL
LIN {X 0,Y 20.33,Z 838.451,A -85,B 0,C 180,E1 889.606,E2 889.606} C_VEL
LIN {X 0,Y 40.886,Z 836.234,A -85,B 0,C 180,E1 888.004,E2 888.004} C_VEL
LIN {X 0,Y 64.658,Z 831.932,A -85,B 0,C 180,E1 886.953,E2 886.953} C_VEL
LIN {X 0,Y 87.466,Z 825.958,A -85,B 0,C 180,E1 886.323,E2 886.323} C_VEL
LIN {X 0,Y 109.265,Z 818.5,A -85,B 0,C 180,E1 885.919,E2 885.919} C_VEL
LIN {X 0,Y 131.074,Z 809.111,A -85,B 0,C 180,E1 885.639,E2 885.639} C_VEL
LIN {X 0,Y 151.382,Z 798.613,A -85,B 0,C 180,E1 885.464,E2 885.464} C_VEL
LIN {X 0,Y 172.586,Z 785.359,A -85,B 0,C 180,E1 885.346,E2 885.346} C_VEL
LIN {X 0,Y 190.21,Z 772.354,A -85,B 0,C 180,E1 885.282,E2 885.282} C_VEL
LIN {X 0,Y 208.845,Z 756.29,A -85,B 0,C 180,E1 885.253,E2 885.253} C_VEL
LIN {X 0,Y 225.39,Z 739.515,A -85,B 0,C 180,E1 885.25,E2 885.25} C_VEL
LIN {X 0,Y 240.878,Z 721.038,A -85,B 0,C 180,E1 885.269,E2 885.269} C_VEL
LIN {X 0,Y 253.765,Z 703.016,A -85,B 0,C 180,E1 885.3,E2 885.3} C_VEL
LIN {X 0,Y 266.121,Z 682.383,A -85,B 0,C 180,E1 885.339,E2 885.339} C_VEL
LIN {X 0,Y 275.883,Z 662.635,A -85,B 0,C 180,E1 885.383,E2 885.383} C_VEL
LIN {X 0,Y 284.339,Z 641.51,A -85,B 0,C 180,E1 885.437,E2 885.437} C_VEL
LIN {X 0,Y 285.935,Z 637.152,A -85,B 0,C 180,E1 885.418,E2 885.418} C_VEL
LIN {X 0,Y 292.758,Z 643.808,A -85,B 0,C 180,E1 879.404,E2 879.404} C_VEL
LIN {X 0,Y 298.278,Z 647.177,A -85,B 0,C 180,E1 875.861,E2 875.861} C_VEL
LIN {X 0,Y 298.597,Z 647.472,A -85,B 0,C 180,E1 875.623,E2 875.623} C_VEL
LIN {X 0,Y 300.145,Z 650.033,A -85,B 0,C 180,E1 874.25,E2 874.25} C_VEL
LIN {X 0,Y 302.552,Z 659.042,A -85,B 0,C 180,E1 870.861,E2 870.861} C_VEL
LIN {X 0,Y 304.085,Z 661.185,A -85,B 0,C 180,E1 869.485,E2 869.485} C_VEL
LIN {X 0,Y 306.708,Z 663.065,A -85,B 0,C 180,E1 867.46,E2 867.46} C_VEL
LIN {X 0,Y 311.111,Z 666.878,A -85,B 0,C 180,E1 863.748,E2 863.748} C_VEL
LIN {X 0,Y 315.591,Z 669.835,A -85,B 0,C 180,E1 859.973,E2 859.973} C_VEL
LIN {X 0,Y 317.612,Z 671.373,A -85,B 0,C 180,E1 858.134,E2 858.134} C_VEL
LIN {X 0,Y 321.415,Z 674.899,A -85,B 0,C 180,E1 854.317,E2 854.317} C_VEL
LIN {X 0,Y 325.281,Z 677.515,A -85,B 0,C 180,E1 850.433,E2 850.433} C_VEL
LIN {X 0,Y 328.23,Z 679.264,A -85,B 0,C 180,E1 847.314,E2 847.314} C_VEL
LIN {X 0,Y 331.143,Z 682.379,A -85,B 0,C 180,E1 843.541,E2 843.541} C_VEL
LIN {X 0,Y 334.1,Z 684.68,A -85,B 0,C 180,E1 839.589,E2 839.589} C_VEL
LIN {X 0,Y 336.852,Z 686.194,A -85,B 0,C 180,E1 835.68,E2 835.68} C_VEL
LIN {X 0,Y 339.215,Z 687.15,A -85,B 0,C 180,E1 831.983,E2 831.983} C_VEL
LIN {X 0,Y 340.888,Z 689.333,A -85,B 0,C 180,E1 828.113,E2 828.113} C_VEL
LIN {X 0,Y 342.169,Z 690.831,A -85,B 0,C 180,E1 824.554,E2 824.554} C_VEL
LIN {X 0,Y 343.242,Z 691.86,A -85,B 0,C 180,E1 820.914,E2 820.914} C_VEL
LIN {X 0,Y 344.096,Z 692.491,A -85,B 0,C 180,E1 817.178,E2 817.178} C_VEL
LIN {X 0,Y 344.64,Z 692.845,A -85,B 0,C 180,E1 813.493,E2 813.493} C_VEL
LIN {X 0,Y 344.743,Z 692.947,A -85,B 0,C 180,E1 809.834,E2 809.834} C_VEL
LIN {X 0,Y 344.536,Z 692.825,A -85,B 0,C 180,E1 806.173,E2 806.173} C_VEL
LIN {X 0,Y 344.077,Z 692.468,A -85,B 0,C 180,E1 802.654,E2 802.654} C_VEL
LIN {X 0,Y 343.246,Z 691.836,A -85,B 0,C 180,E1 798.916,E2 798.916} C_VEL
LIN {X 0,Y 342.101,Z 690.71,A -85,B 0,C 180,E1 795.097,E2 795.097} C_VEL
LIN {X 0,Y 340.636,Z 689.044,A -85,B 0,C 180,E1 791.341,E2 791.341} C_VEL
LIN {X 0,Y 339.054,Z 687.095,A -85,B 0,C 180,E1 787.816,E2 787.816} C_VEL
LIN {X 0,Y 336.717,Z 686.136,A -85,B 0,C 180,E1 784.12,E2 784.12} C_VEL
LIN {X 0,Y 333.954,Z 684.585,A -85,B 0,C 180,E1 780.199,E2 780.199} C_VEL
LIN {X 0,Y 330.828,Z 682.07,A -85,B 0,C 180,E1 776.006,E2 776.006} C_VEL
LIN {X 0,Y 327.586,Z 678.697,A -85,B 0,C 180,E1 771.937,E2 771.937} C_VEL
LIN {X 0,Y 323.929,Z 676.695,A -85,B 0,C 180,E1 768.187,E2 768.187} C_VEL
LIN {X 0,Y 320.141,Z 673.807,A -85,B 0,C 180,E1 764.394,E2 764.394} C_VEL
LIN {X 0,Y 316.281,Z 670.215,A -85,B 0,C 180,E1 760.634,E2 760.634} C_VEL
LIN {X 0,Y 312.025,Z 667.555,A -85,B 0,C 180,E1 757.044,E2 757.044} C_VEL
LIN {X 0,Y 307.64,Z 663.964,A -85,B 0,C 180,E1 753.316,E2 753.316} C_VEL
LIN {X 0,Y 304.985,Z 661.714,A -85,B 0,C 180,E1 751.17,E2 751.17} C_VEL
LIN {X 0,Y 299.534,Z 658.12,A -85,B 0,C 180,E1 747.214,E2 747.214} C_VEL
LIN {X 0,Y 293.9,Z 653.663,A -85,B 0,C 180,E1 743.243,E2 743.243} C_VEL
LIN {X 0,Y 284.904,Z 647.059,A -85,B 0,C 180,E1 736.515,E2 736.515} C_VEL
LIN {X 0,Y 284.473,Z 646.812,A -85,B 0,C 180,E1 736.14,E2 736.14} C_VEL
LIN {X 0,Y 275.975,Z 666.805,A -85,B 0,C 180,E1 736.246,E2 736.246} C_VEL
LIN {X 0,Y 265.2,Z 687.588,A -85,B 0,C 180,E1 736.364,E2 736.364} C_VEL
LIN {X 0,Y 253.369,Z 706.591,A -85,B 0,C 180,E1 736.481,E2 736.481} C_VEL
LIN {X 0,Y 239.464,Z 725.424,A -85,B 0,C 180,E1 736.619,E2 736.619} C_VEL
LIN {X 0,Y 224.504,Z 742.644,A -85,B 0,C 180,E1 736.764,E2 736.764} C_VEL
LIN {X 0,Y 207.975,Z 758.926,A -85,B 0,C 180,E1 736.925,E2 736.925} C_VEL
LIN {X 0,Y 190.388,Z 773.721,A -85,B 0,C 180,E1 737.102,E2 737.102} C_VEL
LIN {X 0,Y 170.705,Z 787.871,A -85,B 0,C 180,E1 737.312,E2 737.312} C_VEL
LIN {X 0,Y 151.006,Z 799.813,A -85,B 0,C 180,E1 737.552,E2 737.552} C_VEL
LIN {X 0,Y 131.292,Z 809.848,A -85,B 0,C 180,E1 737.84,E2 737.84} C_VEL
LIN {X 0,Y 108.323,Z 819.452,A -85,B 0,C 180,E1 738.29,E2 738.29} C_VEL
LIN {X 0,Y 85.643,Z 826.953,A -85,B 0,C 180,E1 738.982,E2 738.982} C_VEL
LIN {X 0,Y 61.856,Z 832.791,A -85,B 0,C 180,E1 740.364,E2 740.364} C_VEL
LIN {X 0,Y 39.284,Z 836.539,A -85,B 0,C 180,E1 743.617,E2 743.617} C_VEL
LIN {X 0,Y 16.606,Z 838.667,A -85,B 0,C 180,E1 758.492,E2 758.492} C_VEL
LIN {X 0,Y 7.999,Z 839.064,A -85,B 0,C 180,E1 810.163,E2 810.163} C_VEL
LIN {X 0,Y 23.254,Z 838.195,A -85,B 0,C 180,E1 869.308,E2 869.308} C_VEL
LIN {X 0,Y 43.36,Z 835.98,A -85,B 0,C 180,E1 877.273,E2 877.273} C_VEL
LIN {X 0,Y 67.018,Z 831.672,A -85,B 0,C 180,E1 880.031,E2 880.031} C_VEL
LIN {X 0,Y 89.852,Z 825.685,A -85,B 0,C 180,E1 881.173,E2 881.173} C_VEL
LIN {X 0,Y 112.027,Z 818.071,A -85,B 0,C 180,E1 881.797,E2 881.797} C_VEL
LIN {X 0,Y 133.368,Z 808.855,A -85,B 0,C 180,E1 882.193,E2 882.193} C_VEL
LIN {X 0,Y 153.08,Z 798.678,A -85,B 0,C 180,E1 882.476,E2 882.476} C_VEL
LIN {X 0,Y 173.812,Z 785.825,A -85,B 0,C 180,E1 882.725,E2 882.725} C_VEL
LIN {X 0,Y 192.457,Z 772.099,A -85,B 0,C 180,E1 882.92,E2 882.92} C_VEL
LIN {X 0,Y 210.041,Z 756.998,A -85,B 0,C 180,E1 883.096,E2 883.096} C_VEL
LIN {X 0,Y 226.569,Z 740.402,A -85,B 0,C 180,E1 883.257,E2 883.257} C_VEL
LIN {X 0,Y 241.527,Z 722.813,A -85,B 0,C 180,E1 883.403,E2 883.403} C_VEL
LIN {X 0,Y 254.911,Z 704.315,A -85,B 0,C 180,E1 883.536,E2 883.536} C_VEL
LIN {X 0,Y 266.739,Z 684.908,A -85,B 0,C 180,E1 883.653,E2 883.653} C_VEL
LIN {X 0,Y 277.001,Z 664.594,A -85,B 0,C 180,E1 883.765,E2 883.765} C_VEL
LIN {X 0,Y 284.559,Z 646.664,A -85,B 0,C 180,E1 883.837,E2 883.837} C_VEL
LIN {X 0,Y 293.002,Z 653.185,A -85,B 0,C 180,E1 877.319,E2 877.319} C_VEL
LIN {X 0,Y 296.106,Z 655.398,A -85,B 0,C 180,E1 875.247,E2 875.247} C_VEL
LIN {X 0,Y 301.6,Z 659.59,A -85,B 0,C 180,E1 871.269,E2 871.269} C_VEL
LIN {X 0,Y 304.085,Z 661.185,A -85,B 0,C 180,E1 869.485,E2 869.485} C_VEL
LIN {X 0,Y 305.438,Z 662.978,A -85,B 0,C 180,E1 868.309,E2 868.309} C_VEL
LIN {X 0,Y 306.505,Z 667.896,A -85,B 0,C 180,E1 866.44,E2 866.44} C_VEL
LIN {X 0,Y 307.382,Z 672.818,A -85,B 0,C 180,E1 864.56,E2 864.56} C_VEL
LIN {X 0,Y 308.477,Z 674.605,A -85,B 0,C 180,E1 863.378,E2 863.378} C_VEL
LIN {X 0,Y 313.317,Z 677.64,A -85,B 0,C 180,E1 859.383,E2 859.383} C_VEL
LIN {X 0,Y 317.421,Z 681.465,A -85,B 0,C 180,E1 855.377,E2 855.377} C_VEL
LIN {X 0,Y 321.193,Z 684.26,A -85,B 0,C 180,E1 851.66,E2 851.66} C_VEL
LIN {X 0,Y 324.976,Z 686.273,A -85,B 0,C 180,E1 847.892,E2 847.892} C_VEL
LIN {X 0,Y 328.021,Z 689.583,A -85,B 0,C 180,E1 843.994,E2 843.994} C_VEL
LIN {X 0,Y 331.165,Z 692.072,A -85,B 0,C 180,E1 839.878,E2 839.878} C_VEL
LIN {X 0,Y 333.772,Z 693.556,A -85,B 0,C 180,E1 836.317,E2 836.317} C_VEL
LIN {X 0,Y 336.322,Z 694.602,A -85,B 0,C 180,E1 832.55,E2 832.55} C_VEL
LIN {X 0,Y 337.414,Z 695.76,A -85,B 0,C 180,E1 830.285,E2 830.285} C_VEL
LIN {X 0,Y 338.975,Z 697.732,A -85,B 0,C 180,E1 826.449,E2 826.449} C_VEL
LIN {X 0,Y 340.163,Z 698.942,A -85,B 0,C 180,E1 822.908,E2 822.908} C_VEL
LIN {X 0,Y 341.192,Z 699.821,A -85,B 0,C 180,E1 819.043,E2 819.043} C_VEL
LIN {X 0,Y 341.907,Z 700.286,A -85,B 0,C 180,E1 815.369,E2 815.369} C_VEL
LIN {X 0,Y 342.222,Z 700.53,A -85,B 0,C 180,E1 811.842,E2 811.842} C_VEL
LIN {X 0,Y 342.205,Z 700.525,A -85,B 0,C 180,E1 808.326,E2 808.326} C_VEL
LIN {X 0,Y 341.946,Z 700.315,A -85,B 0,C 180,E1 804.799,E2 804.799} C_VEL
LIN {X 0,Y 341.261,Z 699.873,A -85,B 0,C 180,E1 801.237,E2 801.237} C_VEL
LIN {X 0,Y 340.318,Z 699.063,A -85,B 0,C 180,E1 797.616,E2 797.616} C_VEL
LIN {X 0,Y 339.112,Z 697.892,A -85,B 0,C 180,E1 793.986,E2 793.986} C_VEL
LIN {X 0,Y 337.567,Z 695.977,A -85,B 0,C 180,E1 790.086,E2 790.086} C_VEL
LIN {X 0,Y 336.406,Z 694.638,A -85,B 0,C 180,E1 787.64,E2 787.64} C_VEL
LIN {X 0,Y 333.901,Z 693.614,A -85,B 0,C 180,E1 783.885,E2 783.885} C_VEL
LIN {X 0,Y 331.2,Z 692.085,A -85,B 0,C 180,E1 780.125,E2 780.125} C_VEL
LIN {X 0,Y 328.025,Z 689.583,A -85,B 0,C 180,E1 776.005,E2 776.005} C_VEL
LIN {X 0,Y 324.993,Z 686.281,A -85,B 0,C 180,E1 772.105,E2 772.105} C_VEL
LIN {X 0,Y 321.346,Z 684.354,A -85,B 0,C 180,E1 768.492,E2 768.492} C_VEL
LIN {X 0,Y 317.636,Z 681.655,A -85,B 0,C 180,E1 764.838,E2 764.838} C_VEL
LIN {X 0,Y 313.715,Z 677.872,A -85,B 0,C 180,E1 760.945,E2 760.945} C_VEL
LIN {X 0,Y 308.915,Z 674.929,A -85,B 0,C 180,E1 757.015,E2 757.015} C_VEL
LIN {X 0,Y 304.441,Z 671.307,A -85,B 0,C 180,E1 753.262,E2 753.262} C_VEL
LIN {X 0,Y 301.752,Z 669.026,A -85,B 0,C 180,E1 751.125,E2 751.125} C_VEL
LIN {X 0,Y 296.152,Z 665.351,A -85,B 0,C 180,E1 747.115,E2 747.115} C_VEL
LIN {X 0,Y 290.715,Z 661.009,A -85,B 0,C 180,E1 743.298,E2 743.298} C_VEL
LIN {X 0,Y 283.102,Z 655.825,A -85,B 0,C 180,E1 737.762,E2 737.762} C_VEL
LIN {X 0,Y 273.218,Z 676.944,A -85,B 0,C 180,E1 737.925,E2 737.925} C_VEL
LIN {X 0,Y 261.941,Z 696.829,A -85,B 0,C 180,E1 738.115,E2 738.115} C_VEL
LIN {X 0,Y 249.104,Z 715.79,A -85,B 0,C 180,E1 738.333,E2 738.333} C_VEL
LIN {X 0,Y 234.71,Z 733.846,A -85,B 0,C 180,E1 738.592,E2 738.592} C_VEL
LIN {X 0,Y 218.23,Z 751.372,A -85,B 0,C 180,E1 738.9,E2 738.9} C_VEL
LIN {X 0,Y 201.22,Z 766.784,A -85,B 0,C 180,E1 739.251,E2 739.251} C_VEL
LIN {X 0,Y 182.63,Z 781.209,A -85,B 0,C 180,E1 739.672,E2 739.672} C_VEL
LIN {X 0,Y 162.997,Z 794.154,A -85,B 0,C 180,E1 740.198,E2 740.198} C_VEL
LIN {X 0,Y 142.325,Z 805.61,A -85,B 0,C 180,E1 740.881,E2 740.881} C_VEL
LIN {X 0,Y 121.663,Z 815.061,A -85,B 0,C 180,E1 741.777,E2 741.777} C_VEL
LIN {X 0,Y 98.972,Z 823.492,A -85,B 0,C 180,E1 743.177,E2 743.177} C_VEL
LIN {X 0,Y 77.036,Z 829.811,A -85,B 0,C 180,E1 745.36,E2 745.36} C_VEL
LIN {X 0,Y 54.658,Z 834.532,A -85,B 0,C 180,E1 749.598,E2 749.598} C_VEL
LIN {X 0,Y 31.897,Z 837.605,A -85,B 0,C 180,E1 761.211,E2 761.211} C_VEL
LIN {X 0,Y 17.862,Z 838.658,A -85,B 0,C 180,E1 792.103,E2 792.103} C_VEL
LIN {X 0,Y 16.073,Z 838.813,A -85,B 0,C 180,E1 810,E2 810} C_VEL
LIN {X 0,Y 28.336,Z 837.94,A -85,B 0,C 180,E1 854.886,E2 854.886} C_VEL
LIN {X 0,Y 47.172,Z 835.726,A -85,B 0,C 180,E1 867.974,E2 867.974} C_VEL
LIN {X 0,Y 70.282,Z 831.412,A -85,B 0,C 180,E1 873.667,E2 873.667} C_VEL
LIN {X 0,Y 92.801,Z 825.449,A -85,B 0,C 180,E1 876.317,E2 876.317} C_VEL
LIN {X 0,Y 114.434,Z 817.982,A -85,B 0,C 180,E1 877.841,E2 877.841} C_VEL
LIN {X 0,Y 136.127,Z 808.598,A -85,B 0,C 180,E1 878.875,E2 878.875} C_VEL
LIN {X 0,Y 156.796,Z 797.839,A -85,B 0,C 180,E1 879.613,E2 879.613} C_VEL
LIN {X 0,Y 177.463,Z 784.855,A -85,B 0,C 180,E1 880.2,E2 880.2} C_VEL
LIN {X 0,Y 195.024,Z 771.844,A -85,B 0,C 180,E1 880.616,E2 880.616} C_VEL
LIN {X 0,Y 212.56,Z 756.743,A -85,B 0,C 180,E1 880.988,E2 880.988} C_VEL
LIN {X 0,Y 228.533,Z 740.717,A -85,B 0,C 180,E1 881.296,E2 881.296} C_VEL
LIN {X 0,Y 243.481,Z 723.204,A -85,B 0,C 180,E1 881.567,E2 881.567} C_VEL
LIN {X 0,Y 257.323,Z 704.069,A -85,B 0,C 180,E1 881.806,E2 881.806} C_VEL
LIN {X 0,Y 269.635,Z 683.762,A -85,B 0,C 180,E1 882.013,E2 882.013} C_VEL
LIN {X 0,Y 279.872,Z 663.237,A -85,B 0,C 180,E1 882.187,E2 882.187} C_VEL
LIN {X 0,Y 283.117,Z 655.839,A -85,B 0,C 180,E1 882.223,E2 882.223} C_VEL
LIN {X 0,Y 291.825,Z 661.874,A -85,B 0,C 180,E1 875.938,E2 875.938} C_VEL
LIN {X 0,Y 296.91,Z 665.912,A -85,B 0,C 180,E1 872.308,E2 872.308} C_VEL
LIN {X 0,Y 302.017,Z 669.177,A -85,B 0,C 180,E1 868.684,E2 868.684} C_VEL
LIN {X 0,Y 306.788,Z 673.332,A -85,B 0,C 180,E1 864.77,E2 864.77} C_VEL
LIN {X 0,Y 308.477,Z 674.605,A -85,B 0,C 180,E1 863.378,E2 863.378} C_VEL
LIN {X 0,Y 309.754,Z 676.668,A -85,B 0,C 180,E1 862.007,E2 862.007} C_VEL
LIN {X 0,Y 311.514,Z 685.702,A -85,B 0,C 180,E1 858.228,E2 858.228} C_VEL
LIN {X 0,Y 312.317,Z 687.104,A -85,B 0,C 180,E1 857.243,E2 857.243} C_VEL
LIN {X 0,Y 316.542,Z 690.627,A -85,B 0,C 180,E1 853.143,E2 853.143} C_VEL
LIN {X 0,Y 320.721,Z 693.111,A -85,B 0,C 180,E1 849.08,E2 849.08} C_VEL
LIN {X 0,Y 322.486,Z 694.356,A -85,B 0,C 180,E1 847.198,E2 847.198} C_VEL
LIN {X 0,Y 325.315,Z 697.292,A -85,B 0,C 180,E1 843.588,E2 843.588} C_VEL
LIN {X 0,Y 328.307,Z 699.569,A -85,B 0,C 180,E1 839.762,E2 839.762} C_VEL
LIN {X 0,Y 331.215,Z 701.163,A -85,B 0,C 180,E1 835.765,E2 835.765} C_VEL
LIN {X 0,Y 333.657,Z 702.151,A -85,B 0,C 180,E1 832.183,E2 832.183} C_VEL
LIN {X 0,Y 335.338,Z 704.251,A -85,B 0,C 180,E1 828.424,E2 828.424} C_VEL
LIN {X 0,Y 336.831,Z 705.913,A -85,B 0,C 180,E1 824.601,E2 824.601} C_VEL
LIN {X 0,Y 337.923,Z 706.949,A -85,B 0,C 180,E1 820.915,E2 820.915} C_VEL
LIN {X 0,Y 338.79,Z 707.593,A -85,B 0,C 180,E1 817.12,E2 817.12} C_VEL
LIN {X 0,Y 339.351,Z 707.944,A -85,B 0,C 180,E1 813.547,E2 813.547} C_VEL
LIN {X 0,Y 339.458,Z 708.051,A -85,B 0,C 180,E1 810,E2 810} C_VEL
LIN {X 0,Y 339.274,Z 707.93,A -85,B 0,C 180,E1 806.283,E2 806.283} C_VEL
LIN {X 0,Y 338.819,Z 707.584,A -85,B 0,C 180,E1 802.71,E2 802.71} C_VEL
LIN {X 0,Y 337.912,Z 706.942,A -85,B 0,C 180,E1 799.084,E2 799.084} C_VEL
LIN {X 0,Y 336.727,Z 705.821,A -85,B 0,C 180,E1 795.205,E2 795.205} C_VEL
LIN {X 0,Y 335.27,Z 704.158,A -85,B 0,C 180,E1 791.392,E2 791.392} C_VEL
LIN {X 0,Y 333.69,Z 702.166,A -85,B 0,C 180,E1 787.801,E2 787.801} C_VEL
LIN {X 0,Y 331.154,Z 701.136,A -85,B 0,C 180,E1 784.126,E2 784.126} C_VEL
LIN {X 0,Y 328.084,Z 699.425,A -85,B 0,C 180,E1 779.941,E2 779.941} C_VEL
LIN {X 0,Y 324.895,Z 696.913,A -85,B 0,C 180,E1 775.878,E2 775.878} C_VEL
LIN {X 0,Y 322.057,Z 693.867,A -85,B 0,C 180,E1 772.296,E2 772.296} C_VEL
LIN {X 0,Y 318.373,Z 691.814,A -85,B 0,C 180,E1 768.641,E2 768.641} C_VEL
LIN {X 0,Y 314.46,Z 689.021,A -85,B 0,C 180,E1 764.844,E2 764.844} C_VEL
LIN {X 0,Y 310.285,Z 685.069,A -85,B 0,C 180,E1 760.779,E2 760.779} C_VEL
LIN {X 0,Y 304.875,Z 681.703,A -85,B 0,C 180,E1 756.413,E2 756.413} C_VEL
LIN {X 0,Y 299.806,Z 677.416,A -85,B 0,C 180,E1 752.249,E2 752.249} C_VEL
LIN {X 0,Y 295.564,Z 674.561,A -85,B 0,C 180,E1 749.152,E2 749.152} C_VEL
LIN {X 0,Y 289.827,Z 670.375,A -85,B 0,C 180,E1 745.108,E2 745.108} C_VEL
LIN {X 0,Y 286.411,Z 667.779,A -85,B 0,C 180,E1 742.799,E2 742.799} C_VEL
LIN {X 0,Y 281.641,Z 664.738,A -85,B 0,C 180,E1 739.393,E2 739.393} C_VEL
LIN {X 0,Y 271.218,Z 685.296,A -85,B 0,C 180,E1 739.629,E2 739.629} C_VEL
LIN {X 0,Y 259.454,Z 704.593,A -85,B 0,C 180,E1 739.902,E2 739.902} C_VEL
LIN {X 0,Y 245.684,Z 723.59,A -85,B 0,C 180,E1 740.238,E2 740.238} C_VEL
LIN {X 0,Y 230.248,Z 741.594,A -85,B 0,C 180,E1 740.644,E2 740.644} C_VEL
LIN {X 0,Y 213.687,Z 758.058,A -85,B 0,C 180,E1 741.118,E2 741.118} C_VEL
LIN {X 0,Y 196.87,Z 772.4,A -85,B 0,C 180,E1 741.66,E2 741.66} C_VEL
LIN {X 0,Y 178.359,Z 786.002,A -85,B 0,C 180,E1 742.34,E2 742.34} C_VEL
LIN {X 0,Y 157.803,Z 798.738,A -85,B 0,C 180,E1 743.262,E2 743.262} C_VEL
LIN {X 0,Y 138.071,Z 808.947,A -85,B 0,C 180,E1 744.379,E2 744.379} C_VEL
LIN {X 0,Y 115.768,Z 818.497,A -85,B 0,C 180,E1 746.078,E2 746.078} C_VEL
LIN {X 0,Y 94.339,Z 825.84,A -85,B 0,C 180,E1 748.485,E2 748.485} C_VEL
LIN {X 0,Y 71.361,Z 831.845,A -85,B 0,C 180,E1 752.791,E2 752.791} C_VEL
LIN {X 0,Y 49.243,Z 835.893,A -85,B 0,C 180,E1 761.301,E2 761.301} C_VEL
LIN {X 0,Y 30.574,Z 838.115,A -85,B 0,C 180,E1 782.004,E2 782.004} C_VEL
LIN {X 0,Y 24.164,Z 838.562,A -85,B 0,C 180,E1 810,E2 810} C_VEL
LIN {X 0,Y 34.642,Z 837.684,A -85,B 0,C 180,E1 845.256,E2 845.256} C_VEL
LIN {X 0,Y 52.968,Z 835.328,A -85,B 0,C 180,E1 860.707,E2 860.707} C_VEL
LIN {X 0,Y 75.326,Z 830.922,A -85,B 0,C 180,E1 868.157,E2 868.157} C_VEL
LIN {X 0,Y 97.972,Z 824.719,A -85,B 0,C 180,E1 872.001,E2 872.001} C_VEL
LIN {X 0,Y 120.879,Z 816.542,A -85,B 0,C 180,E1 874.366,E2 874.366} C_VEL
LIN {X 0,Y 141.761,Z 807.161,A -85,B 0,C 180,E1 875.853,E2 875.853} C_VEL
LIN {X 0,Y 162.94,Z 795.738,A -85,B 0,C 180,E1 876.989,E2 876.989} C_VEL
LIN {X 0,Y 182.472,Z 783.168,A -85,B 0,C 180,E1 877.822,E2 877.822} C_VEL
LIN {X 0,Y 200.98,Z 769.154,A -85,B 0,C 180,E1 878.479,E2 878.479} C_VEL
LIN {X 0,Y 218.442,Z 753.595,A -85,B 0,C 180,E1 879.023,E2 879.023} C_VEL
LIN {X 0,Y 234.354,Z 737.039,A -85,B 0,C 180,E1 879.465,E2 879.465} C_VEL
LIN {X 0,Y 249.214,Z 718.927,A -85,B 0,C 180,E1 879.85,E2 879.85} C_VEL
LIN {X 0,Y 262.522,Z 699.82,A -85,B 0,C 180,E1 880.172,E2 880.172} C_VEL
LIN {X 0,Y 273.766,Z 680.654,A -85,B 0,C 180,E1 880.433,E2 880.433} C_VEL
LIN {X 0,Y 281.684,Z 664.771,A -85,B 0,C 180,E1 880.572,E2 880.572} C_VEL
LIN {X 0,Y 288.159,Z 668.965,A -85,B 0,C 180,E1 876.048,E2 876.048} C_VEL
LIN {X 0,Y 293.943,Z 673.468,A -85,B 0,C 180,E1 872.004,E2 872.004} C_VEL
LIN {X 0,Y 299.333,Z 676.935,A -85,B 0,C 180,E1 868.145,E2 868.145} C_VEL
LIN {X 0,Y 304.131,Z 681.155,A -85,B 0,C 180,E1 864.184,E2 864.184} C_VEL
LIN {X 0,Y 308.828,Z 684.282,A -85,B 0,C 180,E1 860.372,E2 860.372} C_VEL
LIN {X 0,Y 310.993,Z 685.796,A -85,B 0,C 180,E1 858.511,E2 858.511} C_VEL
LIN {X 0,Y 312.317,Z 687.104,A -85,B 0,C 180,E1 857.243,E2 857.243} C_VEL
LIN {X 0,Y 313.308,Z 689.269,A -85,B 0,C 180,E1 855.889,E2 855.889} C_VEL
LIN {X 0,Y 314.194,Z 697.375,A -85,B 0,C 180,E1 852.528,E2 852.528} C_VEL
LIN {X 0,Y 315.183,Z 699.182,A -85,B 0,C 180,E1 851.167,E2 851.167} C_VEL
LIN {X 0,Y 318.732,Z 701.178,A -85,B 0,C 180,E1 847.712,E2 847.712} C_VEL
LIN {X 0,Y 321.735,Z 704.351,A -85,B 0,C 180,E1 843.926,E2 843.926} C_VEL
LIN {X 0,Y 324.765,Z 706.699,A -85,B 0,C 180,E1 840.12,E2 840.12} C_VEL
LIN {X 0,Y 327.95,Z 708.468,A -85,B 0,C 180,E1 835.921,E2 835.921} C_VEL
LIN {X 0,Y 330.474,Z 709.491,A -85,B 0,C 180,E1 832.209,E2 832.209} C_VEL
LIN {X 0,Y 332.23,Z 711.701,A -85,B 0,C 180,E1 828.239,E2 828.239} C_VEL
LIN {X 0,Y 333.729,Z 713.339,A -85,B 0,C 180,E1 824.398,E2 824.398} C_VEL
LIN {X 0,Y 334.792,Z 714.301,A -85,B 0,C 180,E1 821.019,E2 821.019} C_VEL
LIN {X 0,Y 335.68,Z 714.957,A -85,B 0,C 180,E1 817.186,E2 817.186} C_VEL
LIN {X 0,Y 336.254,Z 715.322,A -85,B 0,C 180,E1 813.58,E2 813.58} C_VEL
LIN {X 0,Y 336.371,Z 715.431,A -85,B 0,C 180,E1 810,E2 810} C_VEL
LIN {X 0,Y 336.182,Z 715.31,A -85,B 0,C 180,E1 806.248,E2 806.248} C_VEL
LIN {X 0,Y 335.703,Z 714.948,A -85,B 0,C 180,E1 802.659,E2 802.659} C_VEL
LIN {X 0,Y 334.772,Z 714.29,A -85,B 0,C 180,E1 798.981,E2 798.981} C_VEL
LIN {X 0,Y 333.604,Z 713.201,A -85,B 0,C 180,E1 795.241,E2 795.241} C_VEL
LIN {X 0,Y 332.013,Z 711.415,A -85,B 0,C 180,E1 791.203,E2 791.203} C_VEL
LIN {X 0,Y 330.464,Z 709.487,A -85,B 0,C 180,E1 787.778,E2 787.778} C_VEL
LIN {X 0,Y 328.005,Z 708.49,A -85,B 0,C 180,E1 784.158,E2 784.158} C_VEL
LIN {X 0,Y 324.926,Z 706.801,A -85,B 0,C 180,E1 780.1,E2 780.1} C_VEL
LIN {X 0,Y 322.151,Z 704.713,A -85,B 0,C 180,E1 776.605,E2 776.605} C_VEL
LIN {X 0,Y 318.901,Z 701.373,A -85,B 0,C 180,E1 772.489,E2 772.489} C_VEL
LIN {X 0,Y 315.135,Z 699.148,A -85,B 0,C 180,E1 768.76,E2 768.76} C_VEL
LIN {X 0,Y 310.816,Z 696.104,A -85,B 0,C 180,E1 764.691,E2 764.691} C_VEL
LIN {X 0,Y 306.693,Z 692.215,A -85,B 0,C 180,E1 760.694,E2 760.694} C_VEL
LIN {X 0,Y 301.555,Z 689.054,A -85,B 0,C 180,E1 756.643,E2 756.643} C_VEL
LIN {X 0,Y 296.389,Z 684.799,A -85,B 0,C 180,E1 752.438,E2 752.438} C_VEL
LIN {X 0,Y 293.496,Z 682.682,A -85,B 0,C 180,E1 750.278,E2 750.278} C_VEL
LIN {X 0,Y 287.64,Z 678.691,A -85,B 0,C 180,E1 746.197,E2 746.197} C_VEL
LIN {X 0,Y 282.83,Z 674.936,A -85,B 0,C 180,E1 742.884,E2 742.884} C_VEL
LIN {X 0,Y 280.101,Z 673.532,A -85,B 0,C 180,E1 741.039,E2 741.039} C_VEL
LIN {X 0,Y 269.453,Z 693.05,A -85,B 0,C 180,E1 741.352,E2 741.352} C_VEL
LIN {X 0,Y 256.204,Z 713.223,A -85,B 0,C 180,E1 741.753,E2 741.753} C_VEL
LIN {X 0,Y 241.928,Z 731.5,A -85,B 0,C 180,E1 742.22,E2 742.22} C_VEL
LIN {X 0,Y 226.099,Z 748.787,A -85,B 0,C 180,E1 742.779,E2 742.779} C_VEL
LIN {X 0,Y 209.244,Z 764.506,A -85,B 0,C 180,E1 743.446,E2 743.446} C_VEL
LIN {X 0,Y 190.844,Z 779.211,A -85,B 0,C 180,E1 744.275,E2 744.275} C_VEL
LIN {X 0,Y 172.461,Z 791.757,A -85,B 0,C 180,E1 745.257,E2 745.257} C_VEL
LIN {X 0,Y 153.092,Z 802.951,A -85,B 0,C 180,E1 746.526,E2 746.526} C_VEL
LIN {X 0,Y 131.765,Z 813.23,A -85,B 0,C 180,E1 748.333,E2 748.333} C_VEL
LIN {X 0,Y 110.602,Z 821.635,A -85,B 0,C 180,E1 750.819,E2 750.819} C_VEL
LIN {X 0,Y 87.787,Z 828.696,A -85,B 0,C 180,E1 754.913,E2 754.913} C_VEL
LIN {X 0,Y 66.743,Z 833.568,A -85,B 0,C 180,E1 761.495,E2 761.495} C_VEL
LIN {X 0,Y 46.793,Z 836.832,A -85,B 0,C 180,E1 774.767,E2 774.767} C_VEL
LIN {X 0,Y 34.736,Z 838.075,A -85,B 0,C 180,E1 796.687,E2 796.687} C_VEL
LIN {X 0,Y 32.267,Z 838.31,A -85,B 0,C 180,E1 810,E2 810} C_VEL
LIN {X 0,Y 42.324,Z 837.347,A -85,B 0,C 180,E1 839.742,E2 839.742} C_VEL
LIN {X 0,Y 59.45,Z 834.93,A -85,B 0,C 180,E1 854.939,E2 854.939} C_VEL
LIN {X 0,Y 80.977,Z 830.431,A -85,B 0,C 180,E1 863.376,E2 863.376} C_VEL
LIN {X 0,Y 103.604,Z 823.974,A -85,B 0,C 180,E1 868.13,E2 868.13} C_VEL
LIN {X 0,Y 126.168,Z 815.651,A -85,B 0,C 180,E1 871.092,E2 871.092} C_VEL
LIN {X 0,Y 145.97,Z 806.596,A -85,B 0,C 180,E1 872.929,E2 872.929} C_VEL
LIN {X 0,Y 166.513,Z 795.374,A -85,B 0,C 180,E1 874.384,E2 874.384} C_VEL
LIN {X 0,Y 185.731,Z 782.916,A -85,B 0,C 180,E1 875.473,E2 875.473} C_VEL
LIN {X 0,Y 204.379,Z 768.698,A -85,B 0,C 180,E1 876.349,E2 876.349} C_VEL
LIN {X 0,Y 222.009,Z 752.857,A -85,B 0,C 180,E1 877.069,E2 877.069} C_VEL
LIN {X 0,Y 237.843,Z 736.213,A -85,B 0,C 180,E1 877.641,E2 877.641} C_VEL
LIN {X 0,Y 252.219,Z 718.549,A -85,B 0,C 180,E1 878.122,E2 878.122} C_VEL
LIN {X 0,Y 265.376,Z 699.565,A -85,B 0,C 180,E1 878.528,E2 878.528} C_VEL
LIN {X 0,Y 276.572,Z 680.405,A -85,B 0,C 180,E1 878.858,E2 878.858} C_VEL
LIN {X 0,Y 280.212,Z 673.412,A -85,B 0,C 180,E1 878.935,E2 878.935} C_VEL
LIN {X 0,Y 284.556,Z 676.191,A -85,B 0,C 180,E1 875.946,E2 875.946} C_VEL
LIN {X 0,Y 290.133,Z 680.499,A -85,B 0,C 180,E1 872.051,E2 872.051} C_VEL
LIN {X 0,Y 295.653,Z 684.076,A -85,B 0,C 180,E1 868.159,E2 868.159} C_VEL
LIN {X 0,Y 300.565,Z 688.332,A -85,B 0,C 180,E1 864.163,E2 864.163} C_VEL
LIN {X 0,Y 305.637,Z 691.651,A -85,B 0,C 180,E1 860.119,E2 860.119} C_VEL
LIN {X 0,Y 307.998,Z 693.539,A -85,B 0,C 180,E1 858.02,E2 858.02} C_VEL
LIN {X 0,Y 312.303,Z 697.278,A -85,B 0,C 180,E1 853.917,E2 853.917} C_VEL
LIN {X 0,Y 315.183,Z 699.182,A -85,B 0,C 180,E1 851.167,E2 851.167} C_VEL
LIN {X 0,Y 316.095,Z 700.611,A -85,B 0,C 180,E1 849.997,E2 849.997} C_VEL
LIN {X 0,Y 316.43,Z 704.778,A -85,B 0,C 180,E1 848.116,E2 848.116} C_VEL
LIN {X 0,Y 316.723,Z 709.568,A -85,B 0,C 180,E1 845.936,E2 845.936} C_VEL
LIN {X 0,Y 317.247,Z 710.67,A -85,B 0,C 180,E1 845.05,E2 845.05} C_VEL
LIN {X 0,Y 320.159,Z 713.119,A -85,B 0,C 180,E1 841.435,E2 841.435} C_VEL
LIN {X 0,Y 323.461,Z 715.188,A -85,B 0,C 180,E1 837.224,E2 837.224} C_VEL
LIN {X 0,Y 326.368,Z 716.456,A -85,B 0,C 180,E1 833.209,E2 833.209} C_VEL
LIN {X 0,Y 327.526,Z 717.216,A -85,B 0,C 180,E1 831.301,E2 831.301} C_VEL
LIN {X 0,Y 329.192,Z 719.365,A -85,B 0,C 180,E1 827.499,E2 827.499} C_VEL
LIN {X 0,Y 330.476,Z 720.765,A -85,B 0,C 180,E1 823.788,E2 823.788} C_VEL
LIN {X 0,Y 331.649,Z 721.72,A -85,B 0,C 180,E1 819.895,E2 819.895} C_VEL
LIN {X 0,Y 332.478,Z 722.349,A -85,B 0,C 180,E1 816.215,E2 816.215} C_VEL
LIN {X 0,Y 332.866,Z 722.605,A -85,B 0,C 180,E1 812.582,E2 812.582} C_VEL
LIN {X 0,Y 333.002,Z 722.647,A -85,B 0,C 180,E1 808.968,E2 808.968} C_VEL
LIN {X 0,Y 332.675,Z 722.492,A -85,B 0,C 180,E1 805.518,E2 805.518} C_VEL
LIN {X 0,Y 332.07,Z 722.062,A -85,B 0,C 180,E1 801.865,E2 801.865} C_VEL
LIN {X 0,Y 331.147,Z 721.35,A -85,B 0,C 180,E1 798.329,E2 798.329} C_VEL
LIN {X 0,Y 329.855,Z 720.104,A -85,B 0,C 180,E1 794.349,E2 794.349} C_VEL
LIN {X 0,Y 328.414,Z 718.419,A -85,B 0,C 180,E1 790.699,E2 790.699} C_VEL
LIN {X 0,Y 326.998,Z 716.7,A -85,B 0,C 180,E1 787.719,E2 787.719} C_VEL
LIN {X 0,Y 324.139,Z 715.524,A -85,B 0,C 180,E1 783.629,E2 783.629} C_VEL
LIN {X 0,Y 321.014,Z 713.738,A -85,B 0,C 180,E1 779.629,E2 779.629} C_VEL
LIN {X 0,Y 318.077,Z 711.446,A -85,B 0,C 180,E1 775.978,E2 775.978} C_VEL
LIN {X 0,Y 314.865,Z 708.041,A -85,B 0,C 180,E1 771.955,E2 771.955} C_VEL
LIN {X 0,Y 310.62,Z 705.746,A -85,B 0,C 180,E1 767.97,E2 767.97} C_VEL
LIN {X 0,Y 306.401,Z 702.609,A -85,B 0,C 180,E1 764.033,E2 764.033} C_VEL
LIN {X 0,Y 302.253,Z 698.924,A -85,B 0,C 180,E1 760.17,E2 760.17} C_VEL
LIN {X 0,Y 297.524,Z 695.944,A -85,B 0,C 180,E1 756.5,E2 756.5} C_VEL
LIN {X 0,Y 293.215,Z 692.5,A -85,B 0,C 180,E1 753.065,E2 753.065} C_VEL
LIN {X 0,Y 290.429,Z 690.163,A -85,B 0,C 180,E1 750.861,E2 750.861} C_VEL
LIN {X 0,Y 284.459,Z 686.231,A -85,B 0,C 180,E1 746.738,E2 746.738} C_VEL
LIN {X 0,Y 278.74,Z 681.819,A -85,B 0,C 180,E1 742.72,E2 742.72} C_VEL
LIN {X 0,Y 266.921,Z 701.743,A -85,B 0,C 180,E1 743.133,E2 743.133} C_VEL
LIN {X 0,Y 254.244,Z 719.777,A -85,B 0,C 180,E1 743.611,E2 743.611} C_VEL
LIN {X 0,Y 239.533,Z 737.671,A -85,B 0,C 180,E1 744.212,E2 744.212} C_VEL
LIN {X 0,Y 223.794,Z 754.048,A -85,B 0,C 180,E1 744.915,E2 744.915} C_VEL
LIN {X 0,Y 206.539,Z 769.457,A -85,B 0,C 180,E1 745.789,E2 745.789} C_VEL
LIN {X 0,Y 188.278,Z 783.381,A -85,B 0,C 180,E1 746.856,E2 746.856} C_VEL
LIN {X 0,Y 169.055,Z 795.836,A -85,B 0,C 180,E1 748.21,E2 748.21} C_VEL
LIN {X 0,Y 148.908,Z 806.836,A -85,B 0,C 180,E1 749.985,E2 749.985} C_VEL
LIN {X 0,Y 128.915,Z 816.031,A -85,B 0,C 180,E1 752.288,E2 752.288} C_VEL
LIN {X 0,Y 107.239,Z 824.048,A -85,B 0,C 180,E1 755.793,E2 755.793} C_VEL
LIN {X 0,Y 86.184,Z 830.17,A -85,B 0,C 180,E1 761.055,E2 761.055} C_VEL
LIN {X 0,Y 65.568,Z 834.676,A -85,B 0,C 180,E1 770.175,E2 770.175} C_VEL
LIN {X 0,Y 49.64,Z 837.091,A -85,B 0,C 180,E1 784.977,E2 784.977} C_VEL
LIN {X 0,Y 40.385,Z 838.058,A -85,B 0,C 180,E1 810,E2 810} C_VEL
LIN {X 0,Y 49.674,Z 837.086,A -85,B 0,C 180,E1 835.072,E2 835.072} C_VEL
LIN {X 0,Y 65.568,Z 834.676,A -85,B 0,C 180,E1 849.825,E2 849.825} C_VEL
LIN {X 0,Y 86.184,Z 830.171,A -85,B 0,C 180,E1 858.945,E2 858.945} C_VEL
LIN {X 0,Y 108.214,Z 823.714,A -85,B 0,C 180,E1 864.396,E2 864.396} C_VEL
LIN {X 0,Y 129.91,Z 815.597,A -85,B 0,C 180,E1 867.844,E2 867.844} C_VEL
LIN {X 0,Y 149.912,Z 806.339,A -85,B 0,C 180,E1 870.115,E2 870.115} C_VEL
LIN {X 0,Y 170.066,Z 795.222,A -85,B 0,C 180,E1 871.868,E2 871.868} C_VEL
LIN {X 0,Y 189.292,Z 782.663,A -85,B 0,C 180,E1 873.208,E2 873.208} C_VEL
LIN {X 0,Y 207.553,Z 768.645,A -85,B 0,C 180,E1 874.266,E2 874.266} C_VEL
LIN {X 0,Y 225.172,Z 752.74,A -85,B 0,C 180,E1 875.15,E2 875.15} C_VEL
LIN {X 0,Y 241.057,Z 735.958,A -85,B 0,C 180,E1 875.852,E2 875.852} C_VEL
LIN {X 0,Y 255.26,Z 718.422,A -85,B 0,C 180,E1 876.428,E2 876.428} C_VEL
LIN {X 0,Y 268.444,Z 699.31,A -85,B 0,C 180,E1 876.921,E2 876.921} C_VEL
LIN {X 0,Y 278.754,Z 681.828,A -85,B 0,C 180,E1 877.27,E2 877.27} C_VEL
LIN {X 0,Y 285.607,Z 687.057,A -85,B 0,C 180,E1 872.477,E2 872.477} C_VEL
LIN {X 0,Y 291.528,Z 690.868,A -85,B 0,C 180,E1 868.349,E2 868.349} C_VEL
LIN {X 0,Y 296.527,Z 695.211,A -85,B 0,C 180,E1 864.314,E2 864.314} C_VEL
LIN {X 0,Y 301.435,Z 698.464,A -85,B 0,C 180,E1 860.442,E2 860.442} C_VEL
LIN {X 0,Y 303.664,Z 700.056,A -85,B 0,C 180,E1 858.561,E2 858.561} C_VEL
LIN {X 0,Y 307.931,Z 703.87,A -85,B 0,C 180,E1 854.534,E2 854.534} C_VEL
LIN {X 0,Y 312.476,Z 706.836,A -85,B 0,C 180,E1 850.266,E2 850.266} C_VEL
LIN {X 0,Y 315.301,Z 708.552,A -85,B 0,C 180,E1 847.506,E2 847.506} C_VEL
LIN {X 0,Y 317.247,Z 710.67,A -85,B 0,C 180,E1 845.05,E2 845.05} C_VEL
LIN {X 0,Y 317.916,Z 712.595,A -85,B 0,C 180,E1 843.698,E2 843.698} C_VEL
LIN {X 0,Y 317.764,Z 720.102,A -85,B 0,C 180,E1 840.22,E2 840.22} C_VEL
LIN {X 0,Y 318.376,Z 721.485,A -85,B 0,C 180,E1 838.949,E2 838.949} C_VEL
LIN {X 0,Y 321.335,Z 723.01,A -85,B 0,C 180,E1 835.034,E2 835.034} C_VEL
LIN {X 0,Y 323.712,Z 724.128,A -85,B 0,C 180,E1 831.611,E2 831.611} C_VEL
LIN {X 0,Y 325.281,Z 726.24,A -85,B 0,C 180,E1 827.901,E2 827.901} C_VEL
LIN {X 0,Y 326.694,Z 727.785,A -85,B 0,C 180,E1 823.991,E2 823.991} C_VEL
LIN {X 0,Y 327.951,Z 728.807,A -85,B 0,C 180,E1 820.007,E2 820.007} C_VEL
LIN {X 0,Y 328.844,Z 729.476,A -85,B 0,C 180,E1 816.284,E2 816.284} C_VEL
LIN {X 0,Y 329.252,Z 729.741,A -85,B 0,C 180,E1 812.611,E2 812.611} C_VEL
LIN {X 0,Y 329.394,Z 729.788,A -85,B 0,C 180,E1 808.956,E2 808.956} C_VEL
LIN {X 0,Y 329.055,Z 729.623,A -85,B 0,C 180,E1 805.469,E2 805.469} C_VEL
LIN {X 0,Y 328.409,Z 729.176,A -85,B 0,C 180,E1 801.773,E2 801.773} C_VEL
LIN {X 0,Y 327.462,Z 728.457,A -85,B 0,C 180,E1 798.374,E2 798.374} C_VEL
LIN {X 0,Y 326.096,Z 727.163,A -85,B 0,C 180,E1 794.316,E2 794.316} C_VEL
LIN {X 0,Y 324.558,Z 725.345,A -85,B 0,C 180,E1 790.38,E2 790.38} C_VEL
LIN {X 0,Y 323.285,Z 723.794,A -85,B 0,C 180,E1 787.63,E2 787.63} C_VEL
LIN {X 0,Y 320.212,Z 722.503,A -85,B 0,C 180,E1 783.48,E2 783.48} C_VEL
LIN {X 0,Y 317.432,Z 720.923,A -85,B 0,C 180,E1 779.946,E2 779.946} C_VEL
LIN {X 0,Y 314.149,Z 718.388,A -85,B 0,C 180,E1 775.844,E2 775.844} C_VEL
LIN {X 0,Y 310.624,Z 714.869,A -85,B 0,C 180,E1 771.594,E2 771.594} C_VEL
LIN {X 0,Y 305.973,Z 712.258,A -85,B 0,C 180,E1 767.329,E2 767.329} C_VEL
LIN {X 0,Y 301.857,Z 709.069,A -85,B 0,C 180,E1 763.499,E2 763.499} C_VEL
LIN {X 0,Y 298.13,Z 705.786,A -85,B 0,C 180,E1 760.085,E2 760.085} C_VEL
LIN {X 0,Y 292.79,Z 702.357,A -85,B 0,C 180,E1 755.97,E2 755.97} C_VEL
LIN {X 0,Y 287.85,Z 698.214,A -85,B 0,C 180,E1 752.057,E2 752.057} C_VEL
LIN {X 0,Y 283.128,Z 695.036,A -85,B 0,C 180,E1 748.704,E2 748.704} C_VEL
LIN {X 0,Y 276.887,Z 690.566,A -85,B 0,C 180,E1 744.437,E2 744.437} C_VEL
LIN {X 0,Y 264.665,Z 709.758,A -85,B 0,C 180,E1 744.953,E2 744.953} C_VEL
LIN {X 0,Y 251.053,Z 727.891,A -85,B 0,C 180,E1 745.572,E2 745.572} C_VEL
LIN {X 0,Y 236.004,Z 745.046,A -85,B 0,C 180,E1 746.317,E2 746.317} C_VEL
LIN {X 0,Y 220.295,Z 760.455,A -85,B 0,C 180,E1 747.181,E2 747.181} C_VEL
LIN {X 0,Y 203.185,Z 774.877,A -85,B 0,C 180,E1 748.259,E2 748.259} C_VEL
LIN {X 0,Y 185.108,Z 787.935,A -85,B 0,C 180,E1 749.586,E2 749.586} C_VEL
LIN {X 0,Y 165.126,Z 800.22,A -85,B 0,C 180,E1 751.378,E2 751.378} C_VEL
LIN {X 0,Y 145.3,Z 810.512,A -85,B 0,C 180,E1 753.631,E2 753.631} C_VEL
LIN {X 0,Y 124.771,Z 819.267,A -85,B 0,C 180,E1 756.742,E2 756.742} C_VEL
LIN {X 0,Y 103.804,Z 826.507,A -85,B 0,C 180,E1 761.298,E2 761.298} C_VEL
LIN {X 0,Y 83.857,Z 831.914,A -85,B 0,C 180,E1 768.111,E2 768.111} C_VEL
LIN {X 0,Y 66.7,Z 835.38,A -85,B 0,C 180,E1 778.355,E2 778.355} C_VEL
LIN {X 0,Y 52.313,Z 837.444,A -85,B 0,C 180,E1 797.102,E2 797.102} C_VEL
LIN {X 0,Y 48.517,Z 837.806,A -85,B 0,C 180,E1 810,E2 810} C_VEL
LIN {X 0,Y 57.207,Z 836.834,A -85,B 0,C 180,E1 831.532,E2 831.532} C_VEL
LIN {X 0,Y 72.124,Z 834.421,A -85,B 0,C 180,E1 845.608,E2 845.608} C_VEL
LIN {X 0,Y 92.137,Z 829.837,A -85,B 0,C 180,E1 855.141,E2 855.141} C_VEL
LIN {X 0,Y 113.246,Z 823.454,A -85,B 0,C 180,E1 860.981,E2 860.981} C_VEL
LIN {X 0,Y 134.498,Z 815.342,A -85,B 0,C 180,E1 864.857,E2 864.857} C_VEL
LIN {X 0,Y 154.299,Z 806.032,A -85,B 0,C 180,E1 867.463,E2 867.463} C_VEL
LIN {X 0,Y 174.104,Z 794.964,A -85,B 0,C 180,E1 869.475,E2 869.475} C_VEL
LIN {X 0,Y 193.136,Z 782.408,A -85,B 0,C 180,E1 871.031,E2 871.031} C_VEL
LIN {X 0,Y 211.238,Z 768.39,A -85,B 0,C 180,E1 872.265,E2 872.265} C_VEL
LIN {X 0,Y 228.363,Z 752.829,A -85,B 0,C 180,E1 873.273,E2 873.273} C_VEL
LIN {X 0,Y 243.956,Z 736.318,A -85,B 0,C 180,E1 874.085,E2 874.085} C_VEL
LIN {X 0,Y 258.612,Z 718.17,A -85,B 0,C 180,E1 874.78,E2 874.78} C_VEL
LIN {X 0,Y 271.717,Z 699.055,A -85,B 0,C 180,E1 875.351,E2 875.351} C_VEL
LIN {X 0,Y 276.99,Z 690.49,A -85,B 0,C 180,E1 875.536,E2 875.536} C_VEL
LIN {X 0,Y 283.125,Z 695.04,A -85,B 0,C 180,E1 871.296,E2 871.296} C_VEL
LIN {X 0,Y 287.661,Z 698.022,A -85,B 0,C 180,E1 868.108,E2 868.108} C_VEL
LIN {X 0,Y 292.832,Z 702.377,A -85,B 0,C 180,E1 864.018,E2 864.018} C_VEL
LIN {X 0,Y 298.183,Z 705.806,A -85,B 0,C 180,E1 859.863,E2 859.863} C_VEL
LIN {X 0,Y 302.368,Z 709.508,A -85,B 0,C 180,E1 856.019,E2 856.019} C_VEL
LIN {X 0,Y 306.831,Z 712.804,A -85,B 0,C 180,E1 851.913,E2 851.913} C_VEL
LIN {X 0,Y 311.213,Z 715.323,A -85,B 0,C 180,E1 847.783,E2 847.783} C_VEL
LIN {X 0,Y 314.649,Z 718.813,A -85,B 0,C 180,E1 843.566,E2 843.566} C_VEL
LIN {X 0,Y 318.224,Z 721.398,A -85,B 0,C 180,E1 839.135,E2 839.135} C_VEL
LIN {X 0,Y 318.376,Z 721.485,A -85,B 0,C 180,E1 838.949,E2 838.949} C_VEL
LIN {X 0,Y 319.004,Z 722.96,A -85,B 0,C 180,E1 837.583,E2 837.583} C_VEL
LIN {X 0,Y 318.625,Z 729.672,A -85,B 0,C 180,E1 833.955,E2 833.955} C_VEL
LIN {X 0,Y 319.045,Z 730.636,A -85,B 0,C 180,E1 832.769,E2 832.769} C_VEL
LIN {X 0,Y 320.2,Z 731.81,A -85,B 0,C 180,E1 830.483,E2 830.483} C_VEL
LIN {X 0,Y 321.749,Z 733.755,A -85,B 0,C 180,E1 826.612,E2 826.612} C_VEL
LIN {X 0,Y 323.218,Z 735.125,A -85,B 0,C 180,E1 822.687,E2 822.687} C_VEL
LIN {X 0,Y 324.218,Z 735.959,A -85,B 0,C 180,E1 819.228,E2 819.228} C_VEL
LIN {X 0,Y 324.946,Z 736.442,A -85,B 0,C 180,E1 815.473,E2 815.473} C_VEL
LIN {X 0,Y 325.325,Z 736.715,A -85,B 0,C 180,E1 811.937,E2 811.937} C_VEL
LIN {X 0,Y 325.299,Z 736.705,A -85,B 0,C 180,E1 808.239,E2 808.239} C_VEL
LIN {X 0,Y 325.014,Z 736.487,A -85,B 0,C 180,E1 804.882,E2 804.882} C_VEL
LIN {X 0,Y 324.277,Z 736.015,A -85,B 0,C 180,E1 801.132,E2 801.132} C_VEL
LIN {X 0,Y 323.363,Z 735.246,A -85,B 0,C 180,E1 797.681,E2 797.681} C_VEL
LIN {X 0,Y 321.89,Z 733.885,A -85,B 0,C 180,E1 793.702,E2 793.702} C_VEL
LIN {X 0,Y 320.343,Z 732.019,A -85,B 0,C 180,E1 789.92,E2 789.92} C_VEL
LIN {X 0,Y 319.107,Z 730.655,A -85,B 0,C 180,E1 787.332,E2 787.332} C_VEL
LIN {X 0,Y 316.211,Z 729.428,A -85,B 0,C 180,E1 783.524,E2 783.524} C_VEL
LIN {X 0,Y 313.074,Z 727.623,A -85,B 0,C 180,E1 779.575,E2 779.575} C_VEL
LIN {X 0,Y 309.446,Z 724.713,A -85,B 0,C 180,E1 775.118,E2 775.118} C_VEL
LIN {X 0,Y 306.318,Z 721.642,A -85,B 0,C 180,E1 771.433,E2 771.433} C_VEL
LIN {X 0,Y 301.545,Z 718.914,A -85,B 0,C 180,E1 767.121,E2 767.121} C_VEL
LIN {X 0,Y 297.157,Z 715.456,A -85,B 0,C 180,E1 763.082,E2 763.082} C_VEL
LIN {X 0,Y 293.755,Z 712.494,A -85,B 0,C 180,E1 760.02,E2 760.02} C_VEL
LIN {X 0,Y 288.371,Z 709.017,A -85,B 0,C 180,E1 755.871,E2 755.871} C_VEL
LIN {X 0,Y 282.588,Z 704.09,A -85,B 0,C 180,E1 751.34,E2 751.34} C_VEL
LIN {X 0,Y 276.395,Z 700.113,A -85,B 0,C 180,E1 747.117,E2 747.117} C_VEL
LIN {X 0,Y 274.939,Z 699.221,A -85,B 0,C 180,E1 746.192,E2 746.192} C_VEL
LIN {X 0,Y 262.171,Z 717.918,A -85,B 0,C 180,E1 746.824,E2 746.824} C_VEL
LIN {X 0,Y 247.659,Z 736.02,A -85,B 0,C 180,E1 747.607,E2 747.607} C_VEL
LIN {X 0,Y 232.148,Z 752.574,A -85,B 0,C 180,E1 748.526,E2 748.526} C_VEL
LIN {X 0,Y 215.171,Z 768.136,A -85,B 0,C 180,E1 749.666,E2 749.666} C_VEL
LIN {X 0,Y 197.246,Z 782.151,A -85,B 0,C 180,E1 751.057,E2 751.057} C_VEL
LIN {X 0,Y 178.432,Z 794.706,A -85,B 0,C 180,E1 752.805,E2 752.805} C_VEL
LIN {X 0,Y 157.954,Z 806.255,A -85,B 0,C 180,E1 755.172,E2 755.172} C_VEL
LIN {X 0,Y 138.47,Z 815.518,A -85,B 0,C 180,E1 758.09,E2 758.09} C_VEL
LIN {X 0,Y 117.714,Z 823.529,A -85,B 0,C 180,E1 762.358,E2 762.358} C_VEL
LIN {X 0,Y 97.23,Z 829.825,A -85,B 0,C 180,E1 768.65,E2 768.65} C_VEL
LIN {X 0,Y 79.005,Z 834.166,A -85,B 0,C 180,E1 777.892,E2 777.892} C_VEL
LIN {X 0,Y 64.946,Z 836.577,A -85,B 0,C 180,E1 791.138,E2 791.138} C_VEL
LIN {X 0,Y 56.661,Z 837.553,A -85,B 0,C 180,E1 810,E2 810} C_VEL
LIN {X 0,Y 64.946,Z 836.577,A -85,B 0,C 180,E1 828.862,E2 828.862} C_VEL
LIN {X 0,Y 79.766,Z 834.022,A -85,B 0,C 180,E1 842.614,E2 842.614} C_VEL
LIN {X 0,Y 98.755,Z 829.42,A -85,B 0,C 180,E1 851.929,E2 851.929} C_VEL
LIN {X 0,Y 119.572,Z 822.861,A -85,B 0,C 180,E1 858.09,E2 858.09} C_VEL
LIN {X 0,Y 140.419,Z 814.639,A -85,B 0,C 180,E1 862.239,E2 862.239} C_VEL
LIN {X 0,Y 159.772,Z 805.331,A -85,B 0,C 180,E1 865.063,E2 865.063} C_VEL
LIN {X 0,Y 179.579,Z 793.992,A -85,B 0,C 180,E1 867.311,E2 867.311} C_VEL
LIN {X 0,Y 198.241,Z 781.409,A -85,B 0,C 180,E1 869.025,E2 869.025} C_VEL
LIN {X 0,Y 216.169,Z 767.284,A -85,B 0,C 180,E1 870.406,E2 870.406} C_VEL
LIN {X 0,Y 233.147,Z 751.61,A -85,B 0,C 180,E1 871.537,E2 871.537} C_VEL
LIN {X 0,Y 248.545,Z 735.009,A -85,B 0,C 180,E1 872.443,E2 872.443} C_VEL
LIN {X 0,Y 262.673,Z 717.241,A -85,B 0,C 180,E1 873.201,E2 873.201} C_VEL
LIN {X 0,Y 275.041,Z 699.129,A -85,B 0,C 180,E1 873.788,E2 873.788} C_VEL
LIN {X 0,Y 281.104,Z 703.23,A -85,B 0,C 180,E1 869.664,E2 869.664} C_VEL
LIN {X 0,Y 283.904,Z 705.317,A -85,B 0,C 180,E1 867.635,E2 867.635} C_VEL
LIN {X 0,Y 289.156,Z 709.573,A -85,B 0,C 180,E1 863.505,E2 863.505} C_VEL
LIN {X 0,Y 294.601,Z 712.969,A -85,B 0,C 180,E1 859.335,E2 859.335} C_VEL
LIN {X 0,Y 299.129,Z 717.131,A -85,B 0,C 180,E1 855.121,E2 855.121} C_VEL
LIN {X 0,Y 303.564,Z 720.171,A -85,B 0,C 180,E1 851.039,E2 851.039} C_VEL
LIN {X 0,Y 307.092,Z 722.238,A -85,B 0,C 180,E1 847.704,E2 847.704} C_VEL
LIN {X 0,Y 310.426,Z 725.598,A -85,B 0,C 180,E1 843.641,E2 843.641} C_VEL
LIN {X 0,Y 313.823,Z 728.093,A -85,B 0,C 180,E1 839.566,E2 839.566} C_VEL
LIN {X 0,Y 317.209,Z 729.881,A -85,B 0,C 180,E1 835.226,E2 835.226} C_VEL
LIN {X 0,Y 319.045,Z 730.636,A -85,B 0,C 180,E1 832.769,E2 832.769} C_VEL
LIN {X 0,Y 319.358,Z 731.826,A -85,B 0,C 180,E1 831.498,E2 831.498} C_VEL
LIN {X 0,Y 318.697,Z 735.004,A -85,B 0,C 180,E1 829.895,E2 829.895} C_VEL
LIN {X 0,Y 317.492,Z 739.606,A -85,B 0,C 180,E1 827.613,E2 827.613} C_VEL
LIN {X 0,Y 317.556,Z 740.57,A -85,B 0,C 180,E1 826.618,E2 826.618} C_VEL
LIN {X 0,Y 318.94,Z 741.885,A -85,B 0,C 180,E1 822.676,E2 822.676} C_VEL
LIN {X 0,Y 320.066,Z 742.816,A -85,B 0,C 180,E1 818.805,E2 818.805} C_VEL
LIN {X 0,Y 320.736,Z 743.256,A -85,B 0,C 180,E1 815.187,E2 815.187} C_VEL
LIN {X 0,Y 321.153,Z 743.506,A -85,B 0,C 180,E1 811.427,E2 811.427} C_VEL
LIN {X 0,Y 321.052,Z 743.489,A -85,B 0,C 180,E1 808.037,E2 808.037} C_VEL
LIN {X 0,Y 320.733,Z 743.245,A -85,B 0,C 180,E1 804.454,E2 804.454} C_VEL
LIN {X 0,Y 319.923,Z 742.711,A -85,B 0,C 180,E1 800.829,E2 800.829} C_VEL
LIN {X 0,Y 318.925,Z 741.872,A -85,B 0,C 180,E1 797.139,E2 797.139} C_VEL
LIN {X 0,Y 317.545,Z 740.55,A -85,B 0,C 180,E1 793.35,E2 793.35} C_VEL
LIN {X 0,Y 315.882,Z 738.522,A -85,B 0,C 180,E1 789.431,E2 789.431} C_VEL
LIN {X 0,Y 314.731,Z 737.38,A -85,B 0,C 180,E1 787.197,E2 787.197} C_VEL
LIN {X 0,Y 311.876,Z 736.164,A -85,B 0,C 180,E1 783.439,E2 783.439} C_VEL
LIN {X 0,Y 308.441,Z 734.14,A -85,B 0,C 180,E1 779.192,E2 779.192} C_VEL
LIN {X 0,Y 304.551,Z 730.92,A -85,B 0,C 180,E1 774.508,E2 774.508} C_VEL
LIN {X 0,Y 301.863,Z 728.295,A -85,B 0,C 180,E1 771.416,E2 771.416} C_VEL
LIN {X 0,Y 297.182,Z 725.62,A -85,B 0,C 180,E1 767.176,E2 767.176} C_VEL
LIN {X 0,Y 292.436,Z 721.877,A -85,B 0,C 180,E1 762.874,E2 762.874} C_VEL
LIN {X 0,Y 289.237,Z 719.101,A -85,B 0,C 180,E1 760.014,E2 760.014} C_VEL
LIN {X 0,Y 283.697,Z 715.508,A -85,B 0,C 180,E1 755.806,E2 755.806} C_VEL
LIN {X 0,Y 277.819,Z 710.545,A -85,B 0,C 180,E1 751.215,E2 751.215} C_VEL
LIN {X 0,Y 272.894,Z 707.652,A -85,B 0,C 180,E1 747.996,E2 747.996} C_VEL
LIN {X 0,Y 260.955,Z 724.283,A -85,B 0,C 180,E1 748.67,E2 748.67} C_VEL
LIN {X 0,Y 246.437,Z 741.594,A -85,B 0,C 180,E1 749.57,E2 749.57} C_VEL
LIN {X 0,Y 230.204,Z 758.101,A -85,B 0,C 180,E1 750.688,E2 750.688} C_VEL
LIN {X 0,Y 213.419,Z 772.749,A -85,B 0,C 180,E1 752.01,E2 752.01} C_VEL
LIN {X 0,Y 195.718,Z 786.067,A -85,B 0,C 180,E1 753.624,E2 753.624} C_VEL
LIN {X 0,Y 177.19,Z 798.038,A -85,B 0,C 180,E1 755.654,E2 755.654} C_VEL
LIN {X 0,Y 158.455,Z 808.277,A -85,B 0,C 180,E1 758.198,E2 758.198} C_VEL
LIN {X 0,Y 138.124,Z 817.589,A -85,B 0,C 180,E1 761.791,E2 761.791} C_VEL
LIN {X 0,Y 118.258,Z 825.085,A -85,B 0,C 180,E1 766.645,E2 766.645} C_VEL
LIN {X 0,Y 98.45,Z 831.005,A -85,B 0,C 180,E1 773.912,E2 773.912} C_VEL
LIN {X 0,Y 81.926,Z 834.732,A -85,B 0,C 180,E1 783.938,E2 783.938} C_VEL
LIN {X 0,Y 68.969,Z 836.891,A -85,B 0,C 180,E1 799.137,E2 799.137} C_VEL
LIN {X 0,Y 64.817,Z 837.299,A -85,B 0,C 180,E1 810,E2 810} C_VEL
LIN {X 0,Y 72.799,Z 836.32,A -85,B 0,C 180,E1 826.763,E2 826.763} C_VEL
LIN {X 0,Y 86.861,Z 833.767,A -85,B 0,C 180,E1 839.667,E2 839.667} C_VEL
LIN {X 0,Y 105.074,Z 829.16,A -85,B 0,C 180,E1 848.904,E2 848.904} C_VEL
LIN {X 0,Y 125.261,Z 822.601,A -85,B 0,C 180,E1 855.267,E2 855.267} C_VEL
LIN {X 0,Y 145.607,Z 814.397,A -85,B 0,C 180,E1 859.658,E2 859.658} C_VEL
LIN {X 0,Y 164.642,Z 805.074,A -85,B 0,C 180,E1 862.705,E2 862.705} C_VEL
LIN {X 0,Y 183.998,Z 793.834,A -85,B 0,C 180,E1 865.137,E2 865.137} C_VEL
LIN {X 0,Y 202.589,Z 781.152,A -85,B 0,C 180,E1 867.034,E2 867.034} C_VEL
LIN {X 0,Y 220.496,Z 766.876,A -85,B 0,C 180,E1 868.569,E2 868.569} C_VEL
LIN {X 0,Y 237.639,Z 750.868,A -85,B 0,C 180,E1 869.838,E2 869.838} C_VEL
LIN {X 0,Y 253.02,Z 734.053,A -85,B 0,C 180,E1 870.844,E2 870.844} C_VEL
LIN {X 0,Y 266.923,Z 716.328,A -85,B 0,C 180,E1 871.673,E2 871.673} C_VEL
LIN {X 0,Y 273.065,Z 707.551,A -85,B 0,C 180,E1 871.993,E2 871.993} C_VEL
LIN {X 0,Y 278.64,Z 711.245,A -85,B 0,C 180,E1 868.164,E2 868.164} C_VEL
LIN {X 0,Y 283.949,Z 715.685,A -85,B 0,C 180,E1 863.981,E2 863.981} C_VEL
LIN {X 0,Y 289.225,Z 719.085,A -85,B 0,C 180,E1 859.984,E2 859.984} C_VEL
LIN {X 0,Y 293.171,Z 722.523,A -85,B 0,C 180,E1 856.455,E2 856.455} C_VEL
LIN {X 0,Y 297.661,Z 725.935,A -85,B 0,C 180,E1 852.355,E2 852.355} C_VEL
LIN {X 0,Y 301.947,Z 728.335,A -85,B 0,C 180,E1 848.5,E2 848.5} C_VEL
LIN {X 0,Y 305.201,Z 731.55,A -85,B 0,C 180,E1 844.685,E2 844.685} C_VEL
LIN {X 0,Y 308.688,Z 734.315,A -85,B 0,C 180,E1 840.505,E2 840.505} C_VEL
LIN {X 0,Y 311.92,Z 736.182,A -85,B 0,C 180,E1 836.459,E2 836.459} C_VEL
LIN {X 0,Y 314.751,Z 737.383,A -85,B 0,C 180,E1 832.732,E2 832.732} C_VEL
LIN {X 0,Y 315.959,Z 738.639,A -85,B 0,C 180,E1 830.37,E2 830.37} C_VEL
LIN {X 0,Y 317.556,Z 740.57,A -85,B 0,C 180,E1 826.618,E2 826.618} C_VEL
LIN {X 0,Y 317.591,Z 741.976,A -85,B 0,C 180,E1 825.241,E2 825.241} C_VEL
LIN {X 0,Y 315.268,Z 748.199,A -85,B 0,C 180,E1 821.578,E2 821.578} C_VEL
LIN {X 0,Y 315.119,Z 749.068,A -85,B 0,C 180,E1 820.372,E2 820.372} C_VEL
LIN {X 0,Y 316.09,Z 749.799,A -85,B 0,C 180,E1 816.539,E2 816.539} C_VEL
LIN {X 0,Y 316.556,Z 750.082,A -85,B 0,C 180,E1 812.897,E2 812.897} C_VEL
LIN {X 0,Y 316.747,Z 750.175,A -85,B 0,C 180,E1 809.277,E2 809.277} C_VEL
LIN {X 0,Y 316.385,Z 750.003,A -85,B 0,C 180,E1 805.65,E2 805.65} C_VEL
LIN {X 0,Y 315.801,Z 749.566,A -85,B 0,C 180,E1 802.176,E2 802.176} C_VEL
LIN {X 0,Y 314.695,Z 748.754,A -85,B 0,C 180,E1 798.268,E2 798.268} C_VEL
LIN {X 0,Y 313.44,Z 747.556,A -85,B 0,C 180,E1 794.442,E2 794.442} C_VEL
LIN {X 0,Y 311.825,Z 745.686,A -85,B 0,C 180,E1 790.326,E2 790.326} C_VEL
LIN {X 0,Y 310.376,Z 744.045,A -85,B 0,C 180,E1 787.459,E2 787.459} C_VEL
LIN {X 0,Y 307.217,Z 742.69,A -85,B 0,C 180,E1 783.313,E2 783.313} C_VEL
LIN {X 0,Y 303.742,Z 740.614,A -85,B 0,C 180,E1 779.102,E2 779.102} C_VEL
LIN {X 0,Y 300.522,Z 738.032,A -85,B 0,C 180,E1 775.264,E2 775.264} C_VEL
LIN {X 0,Y 297.373,Z 734.894,A -85,B 0,C 180,E1 771.537,E2 771.537} C_VEL
LIN {X 0,Y 293.098,Z 732.495,A -85,B 0,C 180,E1 767.753,E2 767.753} C_VEL
LIN {X 0,Y 288.503,Z 729.032,A -85,B 0,C 180,E1 763.589,E2 763.589} C_VEL
LIN {X 0,Y 284.782,Z 725.704,A -85,B 0,C 180,E1 760.242,E2 760.242} C_VEL
LIN {X 0,Y 279.113,Z 722.066,A -85,B 0,C 180,E1 755.979,E2 755.979} C_VEL
LIN {X 0,Y 273.905,Z 717.737,A -85,B 0,C 180,E1 751.958,E2 751.958} C_VEL
LIN {X 0,Y 270.881,Z 715.737,A -85,B 0,C 180,E1 749.843,E2 749.843} C_VEL
LIN {X 0,Y 257.077,Z 733.809,A -85,B 0,C 180,E1 750.738,E2 750.738} C_VEL
LIN {X 0,Y 241.838,Z 750.617,A -85,B 0,C 180,E1 751.832,E2 751.832} C_VEL
LIN {X 0,Y 225.676,Z 765.892,A -85,B 0,C 180,E1 753.14,E2 753.14} C_VEL
LIN {X 0,Y 209.111,Z 779.411,A -85,B 0,C 180,E1 754.675,E2 754.675} C_VEL
LIN {X 0,Y 190.743,Z 792.349,A -85,B 0,C 180,E1 756.68,E2 756.68} C_VEL
LIN {X 0,Y 171.66,Z 803.823,A -85,B 0,C 180,E1 759.226,E2 759.226} C_VEL
LIN {X 0,Y 152.597,Z 813.431,A -85,B 0,C 180,E1 762.445,E2 762.445} C_VEL
LIN {X 0,Y 132.941,Z 821.695,A -85,B 0,C 180,E1 766.848,E2 766.848} C_VEL
LIN {X 0,Y 114.113,Z 828.186,A -85,B 0,C 180,E1 772.803,E2 772.803} C_VEL
LIN {X 0,Y 96.99,Z 832.814,A -85,B 0,C 180,E1 781.02,E2 781.02} C_VEL
LIN {X 0,Y 82.295,Z 835.819,A -85,B 0,C 180,E1 793.047,E2 793.047} C_VEL
LIN {X 0,Y 73.96,Z 836.929,A -85,B 0,C 180,E1 806.9,E2 806.9} C_VEL
LIN {X 0,Y 72.989,Z 837.046,A -85,B 0,C 180,E1 810.021,E2 810.021} C_VEL
LIN {X 0,Y 80.797,Z 836.053,A -85,B 0,C 180,E1 825.152,E2 825.152} C_VEL
LIN {X 0,Y 94.149,Z 833.512,A -85,B 0,C 180,E1 837.171,E2 837.171} C_VEL
LIN {X 0,Y 111.652,Z 828.9,A -85,B 0,C 180,E1 846.23,E2 846.23} C_VEL
LIN {X 0,Y 130.347,Z 822.676,A -85,B 0,C 180,E1 852.455,E2 852.455} C_VEL
LIN {X 0,Y 150.176,Z 814.576,A -85,B 0,C 180,E1 857.084,E2 857.084} C_VEL
LIN {X 0,Y 168.828,Z 805.315,A -85,B 0,C 180,E1 860.343,E2 860.343} C_VEL
LIN {X 0,Y 187.865,Z 794.191,A -85,B 0,C 180,E1 862.969,E2 862.969} C_VEL
LIN {X 0,Y 206.198,Z 781.638,A -85,B 0,C 180,E1 865.031,E2 865.031} C_VEL
LIN {X 0,Y 224.186,Z 767.235,A -85,B 0,C 180,E1 866.731,E2 866.731} C_VEL
LIN {X 0,Y 240.369,Z 752.064,A -85,B 0,C 180,E1 868.054,E2 868.054} C_VEL
LIN {X 0,Y 255.396,Z 735.753,A -85,B 0,C 180,E1 869.146,E2 869.146} C_VEL
LIN {X 0,Y 268.41,Z 719.214,A -85,B 0,C 180,E1 870.004,E2 870.004} C_VEL
LIN {X 0,Y 270.955,Z 715.713,A -85,B 0,C 180,E1 870.121,E2 870.121} C_VEL
LIN {X 0,Y 274.195,Z 718.001,A -85,B 0,C 180,E1 867.833,E2 867.833} C_VEL
LIN {X 0,Y 279.787,Z 722.541,A -85,B 0,C 180,E1 863.518,E2 863.518} C_VEL
LIN {X 0,Y 285.361,Z 726.062,A -85,B 0,C 180,E1 859.329,E2 859.329} C_VEL
LIN {X 0,Y 289.993,Z 730.278,A -85,B 0,C 180,E1 855.024,E2 855.024} C_VEL
LIN {X 0,Y 294.98,Z 733.63,A -85,B 0,C 180,E1 850.601,E2 850.601} C_VEL
LIN {X 0,Y 298.123,Z 735.531,A -85,B 0,C 180,E1 847.674,E2 847.674} C_VEL
LIN {X 0,Y 301.686,Z 739.036,A -85,B 0,C 180,E1 843.365,E2 843.365} C_VEL
LIN {X 0,Y 305.021,Z 741.44,A -85,B 0,C 180,E1 839.315,E2 839.315} C_VEL
LIN {X 0,Y 308.09,Z 743.085,A -85,B 0,C 180,E1 835.551,E2 835.551} C_VEL
LIN {X 0,Y 310.796,Z 744.283,A -85,B 0,C 180,E1 831.911,E2 831.911} C_VEL
LIN {X 0,Y 312.419,Z 746.462,A -85,B 0,C 180,E1 828.085,E2 828.085} C_VEL
LIN {X 0,Y 313.923,Z 748.068,A -85,B 0,C 180,E1 824.196,E2 824.196} C_VEL
LIN {X 0,Y 315.119,Z 749.068,A -85,B 0,C 180,E1 820.372,E2 820.372} C_VEL
LIN {X 0,Y 315.041,Z 750.045,A -85,B 0,C 180,E1 819.072,E2 819.072} C_VEL
LIN {X 0,Y 312.923,Z 754.249,A -85,B 0,C 180,E1 816.446,E2 816.446} C_VEL
LIN {X 0,Y 311.776,Z 756.295,A -85,B 0,C 180,E1 814.647,E2 814.647} C_VEL
LIN {X 0,Y 311.694,Z 756.458,A -85,B 0,C 180,E1 814.033,E2 814.033} C_VEL
LIN {X 0,Y 311.872,Z 756.563,A -85,B 0,C 180,E1 810.551,E2 810.551} C_VEL
LIN {X 0,Y 311.793,Z 756.496,A -85,B 0,C 180,E1 807.243,E2 807.243} C_VEL
LIN {X 0,Y 311.259,Z 756.187,A -85,B 0,C 180,E1 803.359,E2 803.359} C_VEL
LIN {X 0,Y 310.458,Z 755.565,A -85,B 0,C 180,E1 799.798,E2 799.798} C_VEL
LIN {X 0,Y 309.103,Z 754.454,A -85,B 0,C 180,E1 795.769,E2 795.769} C_VEL
LIN {X 0,Y 307.702,Z 752.947,A -85,B 0,C 180,E1 792.02,E2 792.02} C_VEL
LIN {X 0,Y 306.002,Z 750.661,A -85,B 0,C 180,E1 787.929,E2 787.929} C_VEL
LIN {X 0,Y 302.84,Z 749.287,A -85,B 0,C 180,E1 783.901,E2 783.901} C_VEL
LIN {X 0,Y 299.757,Z 747.555,A -85,B 0,C 180,E1 780.14,E2 780.14} C_VEL
LIN {X 0,Y 296.111,Z 744.795,A -85,B 0,C 180,E1 775.82,E2 775.82} C_VEL
LIN {X 0,Y 292.756,Z 741.371,A -85,B 0,C 180,E1 771.769,E2 771.769} C_VEL
LIN {X 0,Y 288.063,Z 738.729,A -85,B 0,C 180,E1 767.673,E2 767.673} C_VEL
LIN {X 0,Y 283.4,Z 735.188,A -85,B 0,C 180,E1 763.47,E2 763.47} C_VEL
LIN {X 0,Y 279.545,Z 731.836,A -85,B 0,C 180,E1 760.058,E2 760.058} C_VEL
LIN {X 0,Y 273.791,Z 728.075,A -85,B 0,C 180,E1 755.754,E2 755.754} C_VEL
LIN {X 0,Y 268.544,Z 723.853,A -85,B 0,C 180,E1 751.759,E2 751.759} C_VEL
LIN {X 0,Y 255.484,Z 740.251,A -85,B 0,C 180,E1 752.712,E2 752.712} C_VEL
LIN {X 0,Y 240.9,Z 755.663,A -85,B 0,C 180,E1 753.893,E2 753.893} C_VEL
LIN {X 0,Y 224.287,Z 770.768,A -85,B 0,C 180,E1 755.417,E2 755.417} C_VEL
LIN {X 0,Y 207.186,Z 784.199,A -85,B 0,C 180,E1 757.226,E2 757.226} C_VEL
LIN {X 0,Y 189.16,Z 796.387,A -85,B 0,C 180,E1 759.493,E2 759.493} C_VEL
LIN {X 0,Y 170.754,Z 806.916,A -85,B 0,C 180,E1 762.329,E2 762.329} C_VEL
LIN {X 0,Y 150.883,Z 816.545,A -85,B 0,C 180,E1 766.245,E2 766.245} C_VEL
LIN {X 0,Y 132.332,Z 824.035,A -85,B 0,C 180,E1 771.163,E2 771.163} C_VEL
LIN {X 0,Y 114.563,Z 829.796,A -85,B 0,C 180,E1 777.835,E2 777.835} C_VEL
LIN {X 0,Y 98.333,Z 833.953,A -85,B 0,C 180,E1 787.271,E2 787.271} C_VEL
LIN {X 0,Y 86.438,Z 836.213,A -85,B 0,C 180,E1 799.335,E2 799.335} C_VEL
LIN {X 0,Y 81.161,Z 836.792,A -85,B 0,C 180,E1 810,E2 810} C_VEL
LIN {X 0,Y 89.218,Z 835.725,A -85,B 0,C 180,E1 824.273,E2 824.273} C_VEL
LIN {X 0,Y 102.266,Z 833.098,A -85,B 0,C 180,E1 835.479,E2 835.479} C_VEL
LIN {X 0,Y 119.237,Z 828.409,A -85,B 0,C 180,E1 844.181,E2 844.181} C_VEL
LIN {X 0,Y 137.435,Z 822.082,A -85,B 0,C 180,E1 850.351,E2 850.351} C_VEL
LIN {X 0,Y 155.929,Z 814.32,A -85,B 0,C 180,E1 854.856,E2 854.856} C_VEL
LIN {X 0,Y 174.214,Z 805.059,A -85,B 0,C 180,E1 858.252,E2 858.252} C_VEL
LIN {X 0,Y 192.934,Z 793.933,A -85,B 0,C 180,E1 861.017,E2 861.017} C_VEL
LIN {X 0,Y 211.009,Z 781.381,A -85,B 0,C 180,E1 863.204,E2 863.204} C_VEL
LIN {X 0,Y 228.317,Z 767.373,A -85,B 0,C 180,E1 864.974,E2 864.974} C_VEL
LIN {X 0,Y 244.782,Z 751.809,A -85,B 0,C 180,E1 866.434,E2 866.434} C_VEL
LIN {X 0,Y 259.064,Z 736.028,A -85,B 0,C 180,E1 867.556,E2 867.556} C_VEL
LIN {X 0,Y 268.656,Z 723.743,A -85,B 0,C 180,E1 868.223,E2 868.223} C_VEL
LIN {X 0,Y 274.355,Z 728.476,A -85,B 0,C 180,E1 863.815,E2 863.815} C_VEL
LIN {X 0,Y 280.186,Z 732.184,A -85,B 0,C 180,E1 859.471,E2 859.471} C_VEL
LIN {X 0,Y 284.902,Z 736.449,A -85,B 0,C 180,E1 855.138,E2 855.138} C_VEL
LIN {X 0,Y 289.72,Z 739.752,A -85,B 0,C 180,E1 850.905,E2 850.905} C_VEL
LIN {X 0,Y 293.196,Z 741.835,A -85,B 0,C 180,E1 847.705,E2 847.705} C_VEL
LIN {X 0,Y 297.077,Z 745.587,A -85,B 0,C 180,E1 843.04,E2 843.04} C_VEL
LIN {X 0,Y 300.836,Z 748.2,A -85,B 0,C 180,E1 838.593,E2 838.593} C_VEL
LIN {X 0,Y 304.328,Z 749.982,A -85,B 0,C 180,E1 834.247,E2 834.247} C_VEL
LIN {X 0,Y 306.18,Z 750.922,A -85,B 0,C 180,E1 831.654,E2 831.654} C_VEL
LIN {X 0,Y 307.727,Z 753.012,A -85,B 0,C 180,E1 827.783,E2 827.783} C_VEL
LIN {X 0,Y 309.322,Z 754.65,A -85,B 0,C 180,E1 823.648,E2 823.648} C_VEL
LIN {X 0,Y 310.455,Z 755.565,A -85,B 0,C 180,E1 820.203,E2 820.203} C_VEL
LIN {X 0,Y 311.365,Z 756.239,A -85,B 0,C 180,E1 816.083,E2 816.083} C_VEL
LIN {X 0,Y 311.694,Z 756.458,A -85,B 0,C 180,E1 814.033,E2 814.033} C_VEL
LIN {X 0,Y 311.251,Z 757.233,A -85,B 0,C 180,E1 812.613,E2 812.613} C_VEL
LIN {X 0,Y 309.657,Z 759.484,A -85,B 0,C 180,E1 810.933,E2 810.933} C_VEL
LIN {X 0,Y 307.229,Z 762.372,A -85,B 0,C 180,E1 808.634,E2 808.634} C_VEL
LIN {X 0,Y 306.768,Z 762.749,A -85,B 0,C 180,E1 807.598,E2 807.598} C_VEL
LIN {X 0,Y 306.346,Z 762.486,A -85,B 0,C 180,E1 803.817,E2 803.817} C_VEL
LIN {X 0,Y 305.438,Z 761.79,A -85,B 0,C 180,E1 800.009,E2 800.009} C_VEL
LIN {X 0,Y 304.274,Z 760.856,A -85,B 0,C 180,E1 796.121,E2 796.121} C_VEL
LIN {X 0,Y 302.7,Z 759.209,A -85,B 0,C 180,E1 792.11,E2 792.11} C_VEL
LIN {X 0,Y 300.945,Z 756.867,A -85,B 0,C 180,E1 787.95,E2 787.95} C_VEL
LIN {X 0,Y 298.162,Z 755.666,A -85,B 0,C 180,E1 784.369,E2 784.369} C_VEL
LIN {X 0,Y 294.53,Z 753.648,A -85,B 0,C 180,E1 779.958,E2 779.958} C_VEL
LIN {X 0,Y 290.592,Z 750.584,A -85,B 0,C 180,E1 775.32,E2 775.32} C_VEL
LIN {X 0,Y 287.273,Z 747.358,A -85,B 0,C 180,E1 771.465,E2 771.465} C_VEL
LIN {X 0,Y 282.294,Z 744.443,A -85,B 0,C 180,E1 767.153,E2 767.153} C_VEL
LIN {X 0,Y 277.567,Z 740.71,A -85,B 0,C 180,E1 762.908,E2 762.908} C_VEL
LIN {X 0,Y 274.151,Z 737.817,A -85,B 0,C 180,E1 759.933,E2 759.933} C_VEL
LIN {X 0,Y 268.253,Z 733.899,A -85,B 0,C 180,E1 755.553,E2 755.553} C_VEL
LIN {X 0,Y 265.806,Z 732.171,A -85,B 0,C 180,E1 753.768,E2 753.768} C_VEL
LIN {X 0,Y 251.797,Z 748.767,A -85,B 0,C 180,E1 754.919,E2 754.919} C_VEL
LIN {X 0,Y 237.877,Z 762.732,A -85,B 0,C 180,E1 756.196,E2 756.196} C_VEL
LIN {X 0,Y 220.755,Z 777.415,A -85,B 0,C 180,E1 757.994,E2 757.994} C_VEL
LIN {X 0,Y 203.802,Z 789.991,A -85,B 0,C 180,E1 760.065,E2 760.065} C_VEL
LIN {X 0,Y 185.285,Z 801.704,A -85,B 0,C 180,E1 762.787,E2 762.787} C_VEL
LIN {X 0,Y 167.212,Z 811.429,A -85,B 0,C 180,E1 766.083,E2 766.083} C_VEL
LIN {X 0,Y 148.912,Z 819.821,A -85,B 0,C 180,E1 770.368,E2 770.368} C_VEL
LIN {X 0,Y 130.843,Z 826.617,A -85,B 0,C 180,E1 776.094,E2 776.094} C_VEL
LIN {X 0,Y 114.502,Z 831.572,A -85,B 0,C 180,E1 783.555,E2 783.555} C_VEL
LIN {X 0,Y 100.289,Z 834.959,A -85,B 0,C 180,E1 793.791,E2 793.791} C_VEL
LIN {X 0,Y 91.236,Z 836.324,A -85,B 0,C 180,E1 805.6,E2 805.6} C_VEL
LIN {X 0,Y 89.348,Z 836.538,A -85,B 0,C 180,E1 810,E2 810} C_VEL
LIN {X 0,Y 97.247,Z 835.467,A -85,B 0,C 180,E1 823.073,E2 823.073} C_VEL
LIN {X 0,Y 109.807,Z 832.839,A -85,B 0,C 180,E1 833.618,E2 833.618} C_VEL
LIN {X 0,Y 126.317,Z 828.11,A -85,B 0,C 180,E1 842.118,E2 842.118} C_VEL
LIN {X 0,Y 143.851,Z 821.823,A -85,B 0,C 180,E1 848.213,E2 848.213} C_VEL
LIN {X 0,Y 162.456,Z 813.791,A -85,B 0,C 180,E1 852.912,E2 852.912} C_VEL
LIN {X 0,Y 179.814,Z 804.803,A -85,B 0,C 180,E1 856.29,E2 856.29} C_VEL
LIN {X 0,Y 198.214,Z 793.675,A -85,B 0,C 180,E1 859.168,E2 859.168} C_VEL
LIN {X 0,Y 215.079,Z 781.866,A -85,B 0,C 180,E1 861.35,E2 861.35} C_VEL
LIN {X 0,Y 232.203,Z 767.889,A -85,B 0,C 180,E1 863.236,E2 863.236} C_VEL
LIN {X 0,Y 246.513,Z 754.293,A -85,B 0,C 180,E1 864.611,E2 864.611} C_VEL
LIN {X 0,Y 260.488,Z 738.79,A -85,B 0,C 180,E1 865.807,E2 865.807} C_VEL
LIN {X 0,Y 265.985,Z 732.098,A -85,B 0,C 180,E1 866.197,E2 866.197} C_VEL
LIN {X 0,Y 271.753,Z 736.327,A -85,B 0,C 180,E1 861.821,E2 861.821} C_VEL
LIN {X 0,Y 275.554,Z 738.802,A -85,B 0,C 180,E1 858.946,E2 858.946} C_VEL
LIN {X 0,Y 280.422,Z 743.1,A -85,B 0,C 180,E1 854.512,E2 854.512} C_VEL
LIN {X 0,Y 284.761,Z 745.978,A -85,B 0,C 180,E1 850.675,E2 850.675} C_VEL
LIN {X 0,Y 288.089,Z 748.014,A -85,B 0,C 180,E1 847.649,E2 847.649} C_VEL
LIN {X 0,Y 291.313,Z 751.216,A -85,B 0,C 180,E1 843.78,E2 843.78} C_VEL
LIN {X 0,Y 295.038,Z 753.963,A -85,B 0,C 180,E1 839.431,E2 839.431} C_VEL
LIN {X 0,Y 298.773,Z 755.966,A -85,B 0,C 180,E1 834.918,E2 834.918} C_VEL
LIN {X 0,Y 301.027,Z 756.995,A -85,B 0,C 180,E1 831.839,E2 831.839} C_VEL
LIN {X 0,Y 302.679,Z 759.2,A -85,B 0,C 180,E1 827.891,E2 827.891} C_VEL
LIN {X 0,Y 304.233,Z 760.815,A -85,B 0,C 180,E1 823.881,E2 823.881} C_VEL
LIN {X 0,Y 305.337,Z 761.724,A -85,B 0,C 180,E1 820.375,E2 820.375} C_VEL
LIN {X 0,Y 306.278,Z 762.428,A -85,B 0,C 180,E1 816.372,E2 816.372} C_VEL
LIN {X 0,Y 306.731,Z 762.704,A -85,B 0,C 180,E1 812.99,E2 812.99} C_VEL
LIN {X 0,Y 306.929,Z 762.805,A -85,B 0,C 180,E1 809.253,E2 809.253} C_VEL
LIN {X 0,Y 306.768,Z 762.749,A -85,B 0,C 180,E1 807.598,E2 807.598} C_VEL
LIN {X 0,Y 306.171,Z 763.332,A -85,B 0,C 180,E1 806.26,E2 806.26} C_VEL
LIN {X 0,Y 302.949,Z 766.471,A -85,B 0,C 180,E1 803.651,E2 803.651} C_VEL
LIN {X 0,Y 300.878,Z 768.048,A -85,B 0,C 180,E1 801.798,E2 801.798} C_VEL
LIN {X 0,Y 300.491,Z 768.095,A -85,B 0,C 180,E1 801.055,E2 801.055} C_VEL
LIN {X 0,Y 299.317,Z 767.121,A -85,B 0,C 180,E1 797.264,E2 797.264} C_VEL
LIN {X 0,Y 297.896,Z 765.765,A -85,B 0,C 180,E1 793.223,E2 793.223} C_VEL
LIN {X 0,Y 296.338,Z 763.855,A -85,B 0,C 180,E1 789.458,E2 789.458} C_VEL
LIN {X 0,Y 295.193,Z 762.696,A -85,B 0,C 180,E1 787.287,E2 787.287} C_VEL
LIN {X 0,Y 292.028,Z 761.277,A -85,B 0,C 180,E1 783.332,E2 783.332} C_VEL
LIN {X 0,Y 288.29,Z 758.987,A -85,B 0,C 180,E1 778.885,E2 778.885} C_VEL
LIN {X 0,Y 284.367,Z 755.696,A -85,B 0,C 180,E1 774.292,E2 774.292} C_VEL
LIN {X 0,Y 281.734,Z 753.221,A -85,B 0,C 180,E1 771.331,E2 771.331} C_VEL
LIN {X 0,Y 276.616,Z 750.167,A -85,B 0,C 180,E1 766.899,E2 766.899} C_VEL
LIN {X 0,Y 271.531,Z 746.033,A -85,B 0,C 180,E1 762.366,E2 762.366} C_VEL
LIN {X 0,Y 268.718,Z 743.703,A -85,B 0,C 180,E1 759.962,E2 759.962} C_VEL
LIN {X 0,Y 263.145,Z 740.009,A -85,B 0,C 180,E1 755.843,E2 755.843} C_VEL
LIN {X 0,Y 248.979,Z 755.992,A -85,B 0,C 180,E1 757.144,E2 757.144} C_VEL
LIN {X 0,Y 234.331,Z 770.046,A -85,B 0,C 180,E1 758.665,E2 758.665} C_VEL
LIN {X 0,Y 217.513,Z 783.685,A -85,B 0,C 180,E1 760.672,E2 760.672} C_VEL
LIN {X 0,Y 200.036,Z 795.873,A -85,B 0,C 180,E1 763.135,E2 763.135} C_VEL
LIN {X 0,Y 182.944,Z 806.036,A -85,B 0,C 180,E1 766.046,E2 766.046} C_VEL
LIN {X 0,Y 164.61,Z 815.409,A -85,B 0,C 180,E1 769.937,E2 769.937} C_VEL
LIN {X 0,Y 147.217,Z 822.899,A -85,B 0,C 180,E1 774.74,E2 774.74} C_VEL
LIN {X 0,Y 130.357,Z 828.814,A -85,B 0,C 180,E1 781.105,E2 781.105} C_VEL
LIN {X 0,Y 114.992,Z 833.173,A -85,B 0,C 180,E1 789.648,E2 789.648} C_VEL
LIN {X 0,Y 103.963,Z 835.455,A -85,B 0,C 180,E1 799.471,E2 799.471} C_VEL
LIN {X 0,Y 97.546,Z 836.283,A -85,B 0,C 180,E1 810,E2 810} C_VEL
LIN {X 0,Y 105.318,Z 835.21,A -85,B 0,C 180,E1 822.055,E2 822.055} C_VEL
LIN {X 0,Y 117.645,Z 832.523,A -85,B 0,C 180,E1 832.123,E2 832.123} C_VEL
LIN {X 0,Y 133.29,Z 827.89,A -85,B 0,C 180,E1 840.171,E2 840.171} C_VEL
LIN {X 0,Y 150.453,Z 821.563,A -85,B 0,C 180,E1 846.26,E2 846.26} C_VEL
LIN {X 0,Y 168.064,Z 813.81,A -85,B 0,C 180,E1 850.874,E2 850.874} C_VEL
LIN {X 0,Y 185.61,Z 804.547,A -85,B 0,C 180,E1 854.449,E2 854.449} C_VEL
LIN {X 0,Y 204.217,Z 793.063,A -85,B 0,C 180,E1 857.495,E2 857.495} C_VEL
LIN {X 0,Y 221.228,Z 780.868,A -85,B 0,C 180,E1 859.799,E2 859.799} C_VEL
LIN {X 0,Y 236.464,Z 768.089,A -85,B 0,C 180,E1 861.569,E2 861.569} C_VEL
LIN {X 0,Y 251.384,Z 753.465,A -85,B 0,C 180,E1 863.088,E2 863.088} C_VEL
LIN {X 0,Y 263.158,Z 740.01,A -85,B 0,C 180,E1 864.129,E2 864.129} C_VEL
LIN {X 0,Y 268.843,Z 743.772,A -85,B 0,C 180,E1 859.954,E2 859.954} C_VEL
LIN {X 0,Y 272.818,Z 747.181,A -85,B 0,C 180,E1 856.449,E2 856.449} C_VEL
LIN {X 0,Y 277.827,Z 750.965,A -85,B 0,C 180,E1 852.018,E2 852.018} C_VEL
LIN {X 0,Y 282.3,Z 753.499,A -85,B 0,C 180,E1 848.16,E2 848.16} C_VEL
LIN {X 0,Y 285.526,Z 756.789,A -85,B 0,C 180,E1 844.267,E2 844.267} C_VEL
LIN {X 0,Y 289.117,Z 759.561,A -85,B 0,C 180,E1 840.095,E2 840.095} C_VEL
LIN {X 0,Y 292.626,Z 761.575,A -85,B 0,C 180,E1 835.935,E2 835.935} C_VEL
LIN {X 0,Y 295.659,Z 762.884,A -85,B 0,C 180,E1 832.047,E2 832.047} C_VEL
LIN {X 0,Y 297.311,Z 765.084,A -85,B 0,C 180,E1 828.225,E2 828.225} C_VEL
LIN {X 0,Y 298.868,Z 766.747,A -85,B 0,C 180,E1 824.025,E2 824.025} C_VEL
LIN {X 0,Y 300.016,Z 767.71,A -85,B 0,C 180,E1 820.536,E2 820.536} C_VEL
LIN {X 0,Y 301.02,Z 768.463,A -85,B 0,C 180,E1 816.484,E2 816.484} C_VEL
LIN {X 0,Y 301.512,Z 768.765,A -85,B 0,C 180,E1 813.041,E2 813.041} C_VEL
LIN {X 0,Y 301.698,Z 768.878,A -85,B 0,C 180,E1 809.43,E2 809.43} C_VEL
LIN {X 0,Y 301.35,Z 768.696,A -85,B 0,C 180,E1 805.623,E2 805.623} C_VEL
LIN {X 0,Y 300.729,Z 768.23,A -85,B 0,C 180,E1 802.165,E2 802.165} C_VEL
LIN {X 0,Y 300.491,Z 768.095,A -85,B 0,C 180,E1 801.055,E2 801.055} C_VEL
LIN {X 0,Y 299.42,Z 768.466,A -85,B 0,C 180,E1 799.588,E2 799.588} C_VEL
LIN {X 0,Y 296.535,Z 770.376,A -85,B 0,C 180,E1 797.541,E2 797.541} C_VEL
LIN {X 0,Y 293.62,Z 772.002,A -85,B 0,C 180,E1 795.458,E2 795.458} C_VEL
LIN {X 0,Y 292.779,Z 771.948,A -85,B 0,C 180,E1 794.379,E2 794.379} C_VEL
LIN {X 0,Y 291.147,Z 770.066,A -85,B 0,C 180,E1 790.215,E2 790.215} C_VEL
LIN {X 0,Y 289.84,Z 768.581,A -85,B 0,C 180,E1 787.486,E2 787.486} C_VEL
LIN {X 0,Y 286.379,Z 766.993,A -85,B 0,C 180,E1 783.232,E2 783.232} C_VEL
LIN {X 0,Y 282.662,Z 764.681,A -85,B 0,C 180,E1 778.873,E2 778.873} C_VEL
LIN {X 0,Y 279.142,Z 761.776,A -85,B 0,C 180,E1 774.753,E2 774.753} C_VEL
LIN {X 0,Y 276.321,Z 759.053,A -85,B 0,C 180,E1 771.511,E2 771.511} C_VEL
LIN {X 0,Y 271.555,Z 756.24,A -85,B 0,C 180,E1 767.425,E2 767.425} C_VEL
LIN {X 0,Y 266.358,Z 752.134,A -85,B 0,C 180,E1 762.8,E2 762.8} C_VEL
LIN {X 0,Y 263.363,Z 749.565,A -85,B 0,C 180,E1 760.196,E2 760.196} C_VEL
LIN {X 0,Y 260.265,Z 747.759,A -85,B 0,C 180,E1 758.001,E2 758.001} C_VEL
LIN {X 0,Y 247,Z 762.114,A -85,B 0,C 180,E1 759.362,E2 759.362} C_VEL
LIN {X 0,Y 232.146,Z 775.887,A -85,B 0,C 180,E1 761.088,E2 761.088} C_VEL
LIN {X 0,Y 216.573,Z 788.147,A -85,B 0,C 180,E1 763.162,E2 763.162} C_VEL
LIN {X 0,Y 199.52,Z 799.528,A -85,B 0,C 180,E1 765.849,E2 765.849} C_VEL
LIN {X 0,Y 181.196,Z 810.034,A -85,B 0,C 180,E1 769.374,E2 769.374} C_VEL
LIN {X 0,Y 164.182,Z 818.353,A -85,B 0,C 180,E1 773.501,E2 773.501} C_VEL
LIN {X 0,Y 147.053,Z 825.291,A -85,B 0,C 180,E1 778.949,E2 778.949} C_VEL
LIN {X 0,Y 130.871,Z 830.69,A -85,B 0,C 180,E1 786.114,E2 786.114} C_VEL
LIN {X 0,Y 117.815,Z 834.095,A -85,B 0,C 180,E1 794.747,E2 794.747} C_VEL
LIN {X 0,Y 108.301,Z 835.748,A -85,B 0,C 180,E1 805.234,E2 805.234} C_VEL
LIN {X 0,Y 105.751,Z 836.028,A -85,B 0,C 180,E1 810,E2 810} C_VEL
LIN {X 0,Y 113.422,Z 834.952,A -85,B 0,C 180,E1 821.182,E2 821.182} C_VEL
LIN {X 0,Y 125.177,Z 832.32,A -85,B 0,C 180,E1 830.576,E2 830.576} C_VEL
LIN {X 0,Y 139.805,Z 827.861,A -85,B 0,C 180,E1 838.165,E2 838.165} C_VEL
LIN {X 0,Y 156.42,Z 821.638,A -85,B 0,C 180,E1 844.228,E2 844.228} C_VEL
LIN {X 0,Y 173.56,Z 813.976,A -85,B 0,C 180,E1 848.897,E2 848.897} C_VEL
LIN {X 0,Y 190.712,Z 804.787,A -85,B 0,C 180,E1 852.555,E2 852.555} C_VEL
LIN {X 0,Y 209.341,Z 793.161,A -85,B 0,C 180,E1 855.759,E2 855.759} C_VEL
LIN {X 0,Y 224.785,Z 781.903,A -85,B 0,C 180,E1 857.971,E2 857.971} C_VEL
LIN {X 0,Y 239.554,Z 769.291,A -85,B 0,C 180,E1 859.799,E2 859.799} C_VEL
LIN {X 0,Y 254.036,Z 754.749,A -85,B 0,C 180,E1 861.375,E2 861.375} C_VEL
LIN {X 0,Y 260.386,Z 747.69,A -85,B 0,C 180,E1 861.956,E2 861.956} C_VEL
LIN {X 0,Y 264.8,Z 750.667,A -85,B 0,C 180,E1 858.64,E2 858.64} C_VEL
LIN {X 0,Y 269.585,Z 754.836,A -85,B 0,C 180,E1 854.29,E2 854.29} C_VEL
LIN {X 0,Y 274.746,Z 758.197,A -85,B 0,C 180,E1 849.828,E2 849.828} C_VEL
LIN {X 0,Y 277.278,Z 759.834,A -85,B 0,C 180,E1 847.504,E2 847.504} C_VEL
LIN {X 0,Y 281.141,Z 763.512,A -85,B 0,C 180,E1 842.932,E2 842.932} C_VEL
LIN {X 0,Y 285.164,Z 766.307,A -85,B 0,C 180,E1 838.251,E2 838.251} C_VEL
LIN {X 0,Y 288.5,Z 768.006,A -85,B 0,C 180,E1 834.138,E2 834.138} C_VEL
LIN {X 0,Y 290.372,Z 769.011,A -85,B 0,C 180,E1 831.611,E2 831.611} C_VEL
LIN {X 0,Y 292.132,Z 771.301,A -85,B 0,C 180,E1 827.271,E2 827.271} C_VEL
LIN {X 0,Y 293.521,Z 772.697,A -85,B 0,C 180,E1 823.594,E2 823.594} C_VEL
LIN {X 0,Y 294.868,Z 773.793,A -85,B 0,C 180,E1 819.564,E2 819.564} C_VEL
LIN {X 0,Y 295.636,Z 774.334,A -85,B 0,C 180,E1 815.823,E2 815.823} C_VEL
LIN {X 0,Y 296.091,Z 774.65,A -85,B 0,C 180,E1 812.129,E2 812.129} C_VEL
LIN {X 0,Y 296.084,Z 774.643,A -85,B 0,C 180,E1 808.258,E2 808.258} C_VEL
LIN {X 0,Y 295.74,Z 774.388,A -85,B 0,C 180,E1 804.763,E2 804.763} C_VEL
LIN {X 0,Y 294.978,Z 773.901,A -85,B 0,C 180,E1 800.833,E2 800.833} C_VEL
LIN {X 0,Y 293.742,Z 772.876,A -85,B 0,C 180,E1 797.018,E2 797.018} C_VEL
LIN {X 0,Y 292.779,Z 771.948,A -85,B 0,C 180,E1 794.379,E2 794.379} C_VEL
LIN {X 0,Y 291.608,Z 772.024,A -85,B 0,C 180,E1 792.876,E2 792.876} C_VEL
LIN {X 0,Y 286.934,Z 773.885,A -85,B 0,C 180,E1 789.818,E2 789.818} C_VEL
LIN {X 0,Y 284.306,Z 774.246,A -85,B 0,C 180,E1 787.748,E2 787.748} C_VEL
LIN {X 0,Y 284.122,Z 774.184,A -85,B 0,C 180,E1 787.525,E2 787.525} C_VEL
LIN {X 0,Y 281.003,Z 772.755,A -85,B 0,C 180,E1 783.722,E2 783.722} C_VEL
LIN {X 0,Y 277.608,Z 770.745,A -85,B 0,C 180,E1 779.72,E2 779.72} C_VEL
LIN {X 0,Y 273.778,Z 767.699,A -85,B 0,C 180,E1 775.257,E2 775.257} C_VEL
LIN {X 0,Y 270.601,Z 764.655,A -85,B 0,C 180,E1 771.566,E2 771.566} C_VEL
LIN {X 0,Y 265.164,Z 761.347,A -85,B 0,C 180,E1 766.962,E2 766.962} C_VEL
LIN {X 0,Y 260.227,Z 757.336,A -85,B 0,C 180,E1 762.55,E2 762.55} C_VEL
LIN {X 0,Y 257.527,Z 755.065,A -85,B 0,C 180,E1 760.237,E2 760.237} C_VEL
LIN {X 0,Y 242.211,Z 770.724,A -85,B 0,C 180,E1 762.01,E2 762.01} C_VEL
LIN {X 0,Y 226.777,Z 784.094,A -85,B 0,C 180,E1 764.057,E2 764.057} C_VEL
LIN {X 0,Y 210.756,Z 795.872,A -85,B 0,C 180,E1 766.537,E2 766.537} C_VEL
LIN {X 0,Y 195.159,Z 805.524,A -85,B 0,C 180,E1 769.41,E2 769.41} C_VEL
LIN {X 0,Y 177.621,Z 814.879,A -85,B 0,C 180,E1 773.368,E2 773.368} C_VEL
LIN {X 0,Y 161.037,Z 822.38,A -85,B 0,C 180,E1 778.147,E2 778.147} C_VEL
LIN {X 0,Y 145.105,Z 828.294,A -85,B 0,C 180,E1 784.272,E2 784.272} C_VEL
LIN {X 0,Y 131.231,Z 832.522,A -85,B 0,C 180,E1 791.798,E2 791.798} C_VEL
LIN {X 0,Y 120.632,Z 834.867,A -85,B 0,C 180,E1 800.516,E2 800.516} C_VEL
LIN {X 0,Y 113.984,Z 835.772,A -85,B 0,C 180,E1 810.039,E2 810.039} C_VEL
LIN {X 0,Y 121.547,Z 834.694,A -85,B 0,C 180,E1 820.426,E2 820.426} C_VEL
LIN {X 0,Y 132.972,Z 832.06,A -85,B 0,C 180,E1 829.32,E2 829.32} C_VEL
LIN {X 0,Y 147.169,Z 827.601,A -85,B 0,C 180,E1 836.64,E2 836.64} C_VEL
LIN {X 0,Y 163.34,Z 821.378,A -85,B 0,C 180,E1 842.593,E2 842.593} C_VEL
LIN {X 0,Y 180.07,Z 813.719,A -85,B 0,C 180,E1 847.245,E2 847.245} C_VEL
LIN {X 0,Y 196.866,Z 804.531,A -85,B 0,C 180,E1 850.931,E2 850.931} C_VEL
LIN {X 0,Y 214.13,Z 793.533,A -85,B 0,C 180,E1 854.021,E2 854.021} C_VEL
LIN {X 0,Y 229.482,Z 781.896,A -85,B 0,C 180,E1 856.323,E2 856.323} C_VEL
LIN {X 0,Y 244.955,Z 768.092,A -85,B 0,C 180,E1 858.327,E2 858.327} C_VEL
LIN {X 0,Y 257.579,Z 755.097,A -85,B 0,C 180,E1 859.736,E2 859.736} C_VEL
LIN {X 0,Y 261.946,Z 758.84,A -85,B 0,C 180,E1 855.855,E2 855.855} C_VEL
LIN {X 0,Y 266.688,Z 762.382,A -85,B 0,C 180,E1 851.748,E2 851.748} C_VEL
LIN {X 0,Y 271.303,Z 765.146,A -85,B 0,C 180,E1 847.717,E2 847.717} C_VEL
LIN {X 0,Y 275.029,Z 768.778,A -85,B 0,C 180,E1 843.264,E2 843.264} C_VEL
LIN {X 0,Y 279.056,Z 771.655,A -85,B 0,C 180,E1 838.618,E2 838.618} C_VEL
LIN {X 0,Y 282.764,Z 773.618,A -85,B 0,C 180,E1 834.177,E2 834.177} C_VEL
LIN {X 0,Y 284.603,Z 774.552,A -85,B 0,C 180,E1 831.646,E2 831.646} C_VEL
LIN {X 0,Y 286.4,Z 776.883,A -85,B 0,C 180,E1 827.262,E2 827.262} C_VEL
LIN {X 0,Y 287.804,Z 778.297,A -85,B 0,C 180,E1 823.664,E2 823.664} C_VEL
LIN {X 0,Y 289.124,Z 779.357,A -85,B 0,C 180,E1 819.354,E2 819.354} C_VEL
LIN {X 0,Y 289.859,Z 779.882,A -85,B 0,C 180,E1 815.94,E2 815.94} C_VEL
LIN {X 0,Y 290.321,Z 780.205,A -85,B 0,C 180,E1 812.369,E2 812.369} C_VEL
LIN {X 0,Y 290.369,Z 780.227,A -85,B 0,C 180,E1 808.422,E2 808.422} C_VEL
LIN {X 0,Y 290,Z 779.961,A -85,B 0,C 180,E1 804.857,E2 804.857} C_VEL
LIN {X 0,Y 289.212,Z 779.446,A -85,B 0,C 180,E1 800.85,E2 800.85} C_VEL
LIN {X 0,Y 287.938,Z 778.408,A -85,B 0,C 180,E1 796.751,E2 796.751} C_VEL
LIN {X 0,Y 286.597,Z 777.089,A -85,B 0,C 180,E1 793.169,E2 793.169} C_VEL
LIN {X 0,Y 284.883,Z 774.952,A -85,B 0,C 180,E1 789,E2 789} C_VEL
LIN {X 0,Y 284.122,Z 774.184,A -85,B 0,C 180,E1 787.525,E2 787.525} C_VEL
LIN {X 0,Y 282.181,Z 774.39,A -85,B 0,C 180,E1 786.006,E2 786.006} C_VEL
LIN {X 0,Y 276.792,Z 776.225,A -85,B 0,C 180,E1 783.38,E2 783.38} C_VEL
LIN {X 0,Y 273.108,Z 776.789,A -85,B 0,C 180,E1 781.301,E2 781.301} C_VEL
LIN {X 0,Y 272.36,Z 776.53,A -85,B 0,C 180,E1 780.616,E2 780.616} C_VEL
LIN {X 0,Y 268.906,Z 773.969,A -85,B 0,C 180,E1 776.613,E2 776.613} C_VEL
LIN {X 0,Y 265.552,Z 770.713,A -85,B 0,C 180,E1 772.604,E2 772.604} C_VEL
LIN {X 0,Y 261.975,Z 768.46,A -85,B 0,C 180,E1 769.421,E2 769.421} C_VEL
LIN {X 0,Y 256.697,Z 764.767,A -85,B 0,C 180,E1 764.83,E2 764.83} C_VEL
LIN {X 0,Y 254.142,Z 762.72,A -85,B 0,C 180,E1 762.635,E2 762.635} C_VEL
LIN {X 0,Y 239.501,Z 777.025,A -85,B 0,C 180,E1 764.536,E2 764.536} C_VEL
LIN {X 0,Y 223.786,Z 790.052,A -85,B 0,C 180,E1 766.877,E2 766.877} C_VEL
LIN {X 0,Y 208.253,Z 801.001,A -85,B 0,C 180,E1 769.598,E2 769.598} C_VEL
LIN {X 0,Y 192.396,Z 810.396,A -85,B 0,C 180,E1 772.928,E2 772.928} C_VEL
LIN {X 0,Y 176.177,Z 818.576,A -85,B 0,C 180,E1 777.134,E2 777.134} C_VEL
LIN {X 0,Y 160.871,Z 825.014,A -85,B 0,C 180,E1 782.217,E2 782.217} C_VEL
LIN {X 0,Y 145.581,Z 830.352,A -85,B 0,C 180,E1 789.076,E2 789.076} C_VEL
LIN {X 0,Y 133.383,Z 833.709,A -85,B 0,C 180,E1 797.004,E2 797.004} C_VEL
LIN {X 0,Y 124.429,Z 835.268,A -85,B 0,C 180,E1 806.314,E2 806.314} C_VEL
LIN {X 0,Y 122.187,Z 835.518,A -85,B 0,C 180,E1 810,E2 810} C_VEL
LIN {X 0,Y 129.697,Z 834.436,A -85,B 0,C 180,E1 819.764,E2 819.764} C_VEL
LIN {X 0,Y 140.828,Z 831.801,A -85,B 0,C 180,E1 828.203,E2 828.203} C_VEL
LIN {X 0,Y 154.63,Z 827.341,A -85,B 0,C 180,E1 835.262,E2 835.262} C_VEL
LIN {X 0,Y 170.589,Z 821.026,A -85,B 0,C 180,E1 841.159,E2 841.159} C_VEL
LIN {X 0,Y 186.716,Z 813.461,A -85,B 0,C 180,E1 845.709,E2 845.709} C_VEL
LIN {X 0,Y 203.172,Z 804.22,A -85,B 0,C 180,E1 849.407,E2 849.407} C_VEL
LIN {X 0,Y 219.423,Z 793.317,A -85,B 0,C 180,E1 852.406,E2 852.406} C_VEL
LIN {X 0,Y 234.375,Z 781.463,A -85,B 0,C 180,E1 854.739,E2 854.739} C_VEL
LIN {X 0,Y 248.713,Z 768.285,A -85,B 0,C 180,E1 856.688,E2 856.688} C_VEL
LIN {X 0,Y 254.253,Z 762.637,A -85,B 0,C 180,E1 857.338,E2 857.338} C_VEL
LIN {X 0,Y 259.034,Z 766.555,A -85,B 0,C 180,E1 853.094,E2 853.094} C_VEL
LIN {X 0,Y 264.435,Z 769.868,A -85,B 0,C 180,E1 848.493,E2 848.493} C_VEL
LIN {X 0,Y 267.165,Z 772.416,A -85,B 0,C 180,E1 845.455,E2 845.455} C_VEL
LIN {X 0,Y 271.158,Z 775.731,A -85,B 0,C 180,E1 840.779,E2 840.779} C_VEL
LIN {X 0,Y 275.184,Z 778.184,A -85,B 0,C 180,E1 836.08,E2 836.08} C_VEL
LIN {X 0,Y 278.184,Z 779.54,A -85,B 0,C 180,E1 832.394,E2 832.394} C_VEL
LIN {X 0,Y 279.936,Z 781.577,A -85,B 0,C 180,E1 828.751,E2 828.751} C_VEL
LIN {X 0,Y 281.475,Z 783.267,A -85,B 0,C 180,E1 824.608,E2 824.608} C_VEL
LIN {X 0,Y 282.841,Z 784.464,A -85,B 0,C 180,E1 820.592,E2 820.592} C_VEL
LIN {X 0,Y 283.833,Z 785.195,A -85,B 0,C 180,E1 816.472,E2 816.472} C_VEL
LIN {X 0,Y 284.349,Z 785.53,A -85,B 0,C 180,E1 813.003,E2 813.003} C_VEL
LIN {X 0,Y 284.554,Z 785.651,A -85,B 0,C 180,E1 808.993,E2 808.993} C_VEL
LIN {X 0,Y 284.12,Z 785.386,A -85,B 0,C 180,E1 805.155,E2 805.155} C_VEL
LIN {X 0,Y 283.426,Z 784.899,A -85,B 0,C 180,E1 801.684,E2 801.684} C_VEL
LIN {X 0,Y 282.255,Z 783.964,A -85,B 0,C 180,E1 797.521,E2 797.521} C_VEL
LIN {X 0,Y 280.755,Z 782.548,A -85,B 0,C 180,E1 793.447,E2 793.447} C_VEL
LIN {X 0,Y 279.236,Z 780.71,A -85,B 0,C 180,E1 789.677,E2 789.677} C_VEL
LIN {X 0,Y 278.132,Z 779.532,A -85,B 0,C 180,E1 787.501,E2 787.501} C_VEL
LIN {X 0,Y 274.852,Z 778.017,A -85,B 0,C 180,E1 783.495,E2 783.495} C_VEL
LIN {X 0,Y 272.36,Z 776.53,A -85,B 0,C 180,E1 780.616,E2 780.616} C_VEL
LIN {X 0,Y 270.027,Z 776.309,A -85,B 0,C 180,E1 778.93,E2 778.93} C_VEL
LIN {X 0,Y 261.987,Z 777.26,A -85,B 0,C 180,E1 774.947,E2 774.947} C_VEL
LIN {X 0,Y 260.027,Z 776.506,A -85,B 0,C 180,E1 773.425,E2 773.425} C_VEL
LIN {X 0,Y 258.066,Z 774.863,A -85,B 0,C 180,E1 771.408,E2 771.408} C_VEL
LIN {X 0,Y 253.109,Z 771.808,A -85,B 0,C 180,E1 767.201,E2 767.201} C_VEL
LIN {X 0,Y 250.596,Z 770.191,A -85,B 0,C 180,E1 765.182,E2 765.182} C_VEL
LIN {X 0,Y 236.822,Z 783.012,A -85,B 0,C 180,E1 767.178,E2 767.178} C_VEL
LIN {X 0,Y 222.192,Z 794.765,A -85,B 0,C 180,E1 769.611,E2 769.611} C_VEL
LIN {X 0,Y 206.344,Z 805.602,A -85,B 0,C 180,E1 772.722,E2 772.722} C_VEL
LIN {X 0,Y 190.859,Z 814.464,A -85,B 0,C 180,E1 776.403,E2 776.403} C_VEL
LIN {X 0,Y 175.336,Z 821.861,A -85,B 0,C 180,E1 781.007,E2 781.007} C_VEL
LIN {X 0,Y 160.861,Z 827.543,A -85,B 0,C 180,E1 786.56,E2 786.56} C_VEL
LIN {X 0,Y 147.626,Z 831.868,A -85,B 0,C 180,E1 793.474,E2 793.474} C_VEL
LIN {X 0,Y 137.03,Z 834.342,A -85,B 0,C 180,E1 801.609,E2 801.609} C_VEL
LIN {X 0,Y 130.417,Z 835.262,A -85,B 0,C 180,E1 810,E2 810} C_VEL
LIN {X 0,Y 137.865,Z 834.178,A -85,B 0,C 180,E1 819.181,E2 819.181} C_VEL
LIN {X 0,Y 148.732,Z 831.541,A -85,B 0,C 180,E1 827.205,E2 827.205} C_VEL
LIN {X 0,Y 161.789,Z 827.216,A -85,B 0,C 180,E1 833.846,E2 833.846} C_VEL
LIN {X 0,Y 177.522,Z 820.86,A -85,B 0,C 180,E1 839.711,E2 839.711} C_VEL
LIN {X 0,Y 192.71,Z 813.51,A -85,B 0,C 180,E1 844.079,E2 844.079} C_VEL
LIN {X 0,Y 208.806,Z 804.023,A -85,B 0,C 180,E1 847.8,E2 847.8} C_VEL
LIN {X 0,Y 223.894,Z 793.44,A -85,B 0,C 180,E1 850.691,E2 850.691} C_VEL
LIN {X 0,Y 237.695,Z 782.263,A -85,B 0,C 180,E1 852.955,E2 852.955} C_VEL
LIN {X 0,Y 250.747,Z 770.003,A -85,B 0,C 180,E1 854.824,E2 854.824} C_VEL
LIN {X 0,Y 255.95,Z 773.657,A -85,B 0,C 180,E1 850.381,E2 850.381} C_VEL
LIN {X 0,Y 259.308,Z 775.722,A -85,B 0,C 180,E1 847.41,E2 847.41} C_VEL
LIN {X 0,Y 263.144,Z 779.399,A -85,B 0,C 180,E1 842.889,E2 842.889} C_VEL
LIN {X 0,Y 267.022,Z 782.129,A -85,B 0,C 180,E1 838.364,E2 838.364} C_VEL
LIN {X 0,Y 270.549,Z 784.036,A -85,B 0,C 180,E1 834.218,E2 834.218} C_VEL
LIN {X 0,Y 272.608,Z 785.162,A -85,B 0,C 180,E1 831.516,E2 831.516} C_VEL
LIN {X 0,Y 274.144,Z 787.155,A -85,B 0,C 180,E1 827.62,E2 827.62} C_VEL
LIN {X 0,Y 275.78,Z 788.826,A -85,B 0,C 180,E1 823.417,E2 823.417} C_VEL
LIN {X 0,Y 277.048,Z 789.85,A -85,B 0,C 180,E1 819.346,E2 819.346} C_VEL
LIN {X 0,Y 277.786,Z 790.385,A -85,B 0,C 180,E1 815.991,E2 815.991} C_VEL
LIN {X 0,Y 278.301,Z 790.736,A -85,B 0,C 180,E1 812.059,E2 812.059} C_VEL
LIN {X 0,Y 278.265,Z 790.71,A -85,B 0,C 180,E1 808.147,E2 808.147} C_VEL
LIN {X 0,Y 277.903,Z 790.44,A -85,B 0,C 180,E1 804.633,E2 804.633} C_VEL
LIN {X 0,Y 277.126,Z 789.927,A -85,B 0,C 180,E1 800.866,E2 800.866} C_VEL
LIN {X 0,Y 275.733,Z 788.775,A -85,B 0,C 180,E1 796.581,E2 796.581} C_VEL
LIN {X 0,Y 274.301,Z 787.328,A -85,B 0,C 180,E1 792.749,E2 792.749} C_VEL
LIN {X 0,Y 272.671,Z 785.247,A -85,B 0,C 180,E1 788.653,E2 788.653} C_VEL
LIN {X 0,Y 270.923,Z 784.207,A -85,B 0,C 180,E1 786.242,E2 786.242} C_VEL
LIN {X 0,Y 267.332,Z 782.32,A -85,B 0,C 180,E1 781.966,E2 781.966} C_VEL
LIN {X 0,Y 263.369,Z 779.562,A -85,B 0,C 180,E1 777.379,E2 777.379} C_VEL
LIN {X 0,Y 260.027,Z 776.506,A -85,B 0,C 180,E1 773.425,E2 773.425} C_VEL
LIN {X 0,Y 258.566,Z 776.204,A -85,B 0,C 180,E1 772.501,E2 772.501} C_VEL
LIN {X 0,Y 254.504,Z 777.133,A -85,B 0,C 180,E1 771.09,E2 771.09} C_VEL
LIN {X 0,Y 249.835,Z 778.086,A -85,B 0,C 180,E1 769.503,E2 769.503} C_VEL
LIN {X 0,Y 248.404,Z 777.777,A -85,B 0,C 180,E1 768.699,E2 768.699} C_VEL
LIN {X 0,Y 247.251,Z 777.143,A -85,B 0,C 180,E1 767.835,E2 767.835} C_VEL
LIN {X 0,Y 233.222,Z 789.562,A -85,B 0,C 180,E1 770.121,E2 770.121} C_VEL
LIN {X 0,Y 218.663,Z 800.679,A -85,B 0,C 180,E1 772.874,E2 772.874} C_VEL
LIN {X 0,Y 204.281,Z 810.055,A -85,B 0,C 180,E1 776.085,E2 776.085} C_VEL
LIN {X 0,Y 189.847,Z 818.027,A -85,B 0,C 180,E1 779.979,E2 779.979} C_VEL
LIN {X 0,Y 175.711,Z 824.476,A -85,B 0,C 180,E1 784.738,E2 784.738} C_VEL
